# B&R Automation Studio project NewPendant_NG4_11_05_25A (part 8)

```c
					break;

			}

			if (Process[m->pCfg->HeadCfg.OSC.PROC_Indx].Param[1] == 0)
			{

				if(1)
				{

					curCalib->Points[CALIB_OSC_SFT_LIMIT].val[1] = TML_MTR_INST[m->pCfg->HeadCfg.OSC.TML_A_Indx].PosFBK + OSC_TML_Param_Set[0].MaxOscAmpl/2.0 ;

					if (m->pCfg->HeadCfg.OSC.TML_A_Indx == m->pCfg->HeadCfg.OSC.TML_B_Indx) // Only One OSC
						curCalib->Points[CALIB_OSC_SFT_LIMIT].val[3] = curCalib->Points[CALIB_OSC_SFT_LIMIT].val[1];

					strcpy(hmi->pMessage[0], " OSC Positive  ");
					strcpy(hmi->pMessage[1], " Software  ");
					strcpy(hmi->pMessage[2], " Limit SET ");
					strcpy(hmi->pMessage[3], " ");
					TimerStart(&hmi->MsgTmr, 1.5);

				}
				else
				{
					strcpy(hmi->pMessage[0], " Positive is ");
					strcpy(hmi->pMessage[1], "	 lower ");
					strcpy(hmi->pMessage[2], " than negative");
					strcpy(hmi->pMessage[3], "	TRY AGAIN ");
					TimerStart(&hmi->MsgTmr, 2.0);

				}

			}
			else
			{

				//if (TML_MTR_INST[m->pCfg->HeadCfg.OSC.TML_B_Indx].PosFBK > curCalib->Points[CALIB_OSC_SFT_LIMIT].val[2])
				if(1)
				{
					curCalib->Points[CALIB_OSC_SFT_LIMIT].val[3] = TML_MTR_INST[m->pCfg->HeadCfg.OSC.TML_B_Indx].PosFBK + OSC_TML_Param_Set[0].MaxOscAmpl/2.0;

					if (m->pCfg->HeadCfg.OSC.TML_A_Indx == m->pCfg->HeadCfg.OSC.TML_B_Indx) // Only One OSC
						curCalib->Points[CALIB_OSC_SFT_LIMIT].val[1] = curCalib->Points[CALIB_OSC_SFT_LIMIT].val[3];

					strcpy(hmi->pMessage[0], " OSC Positive  ");
					strcpy(hmi->pMessage[1], " Software  ");
					strcpy(hmi->pMessage[2], " Limit SET ");
					strcpy(hmi->pMessage[3], " ");
					TimerStart(&hmi->MsgTmr, 1.5);

				}
				else
				{
					strcpy(hmi->pMessage[0], " Positive is ");
					strcpy(hmi->pMessage[1], "	 lower ");
					strcpy(hmi->pMessage[2], " than negative");
					strcpy(hmi->pMessage[3], "	TRY AGAIN ");
					TimerStart(&hmi->MsgTmr, 2.0);

				}

			}

		break;

		/////////////////////////////////////////////////////////////////////////
		case EVNT_OSC_NEG_LIMIT_SET:

			if (m->pCfg->HeadCfg.OSC.Limits_Harcoded)
			{

				strcpy(hmi->pMessage[0], " OSC Limits  ");
				strcpy(hmi->pMessage[1], " are hardcoded  ");
				strcpy(hmi->pMessage[2], " Operation ");
				strcpy(hmi->pMessage[3], " denied");
				TimerStart(&hmi->MsgTmr, 1.5);

				break;

			}

			if((curCalib->GenSetup[SETUP_HEAD_SETUP] == BPV_v2_MT_BO_TOS)
				|| (curCalib->GenSetup[SETUP_HEAD_SETUP] == BPV_v2_TT_BO_TOS)
				|| (curCalib->GenSetup[SETUP_HEAD_SETUP] == BPV_v2_MPGH)
				|| (curCalib->GenSetup[SETUP_HEAD_SETUP] == BPV_v2_MPGV)
				 ){

					curCalib->Points[CALIB_OSC_SFT_LIMIT].val[0] = TML_MTR_INST[m->pCfg->HeadCfg.TVL.TML_Indx].PosFBK;

					strcpy(hmi->pMessage[0], " TVL (OSC) Negative  ");
					strcpy(hmi->pMessage[1], " Software  ");
					strcpy(hmi->pMessage[2], " Limit SET ");
					strcpy(hmi->pMessage[3], " ");
					TimerStart(&hmi->MsgTmr, 1.5);

					break;

			}

			if (Process[m->pCfg->HeadCfg.OSC.PROC_Indx].Param[1] == 0)
			{

				//if (TML_MTR_INST[m->pCfg->HeadCfg.OSC.TML_A_Indx].PosFBK < curCalib->Points[CALIB_OSC_SFT_LIMIT].val[1])
				if(1)
				{
					curCalib->Points[CALIB_OSC_SFT_LIMIT].val[0] = TML_MTR_INST[m->pCfg->HeadCfg.OSC.TML_A_Indx].PosFBK - OSC_TML_Param_Set[0].MaxOscAmpl/2.0;

					if (m->pCfg->HeadCfg.OSC.TML_A_Indx == m->pCfg->HeadCfg.OSC.TML_B_Indx) // Only One OSC
						curCalib->Points[CALIB_OSC_SFT_LIMIT].val[2] = curCalib->Points[CALIB_OSC_SFT_LIMIT].val[0];

					strcpy(hmi->pMessage[0], " OSC Negative  ");
					strcpy(hmi->pMessage[1], " Software  ");
					strcpy(hmi->pMessage[2], " Limit SET ");
					strcpy(hmi->pMessage[3], " ");
					TimerStart(&hmi->MsgTmr, 1.5);

				}
				else
				{
					strcpy(hmi->pMessage[0], " Negative is ");
					strcpy(hmi->pMessage[1], "	 greater ");
					strcpy(hmi->pMessage[2], " than positive");
					strcpy(hmi->pMessage[3], "	TRY AGAIN ");
					TimerStart(&hmi->MsgTmr, 2.0);

				}
			}
			else
			{

				//if (TML_MTR_INST[m->pCfg->HeadCfg.OSC.TML_B_Indx].PosFBK < curCalib->Points[CALIB_OSC_SFT_LIMIT].val[3])
				if(1)
				{
					curCalib->Points[CALIB_OSC_SFT_LIMIT].val[2] = TML_MTR_INST[m->pCfg->HeadCfg.OSC.TML_B_Indx].PosFBK - OSC_TML_Param_Set[0].MaxOscAmpl/2.0;

					if (m->pCfg->HeadCfg.OSC.TML_A_Indx == m->pCfg->HeadCfg.OSC.TML_B_Indx) // Only One OSC
						curCalib->Points[CALIB_OSC_SFT_LIMIT].val[0] = curCalib->Points[CALIB_OSC_SFT_LIMIT].val[2];

					strcpy(hmi->pMessage[0], " OSC Negative  ");
					strcpy(hmi->pMessage[1], " Software  ");
					strcpy(hmi->pMessage[2], " Limit SET ");
					strcpy(hmi->pMessage[3], " ");
					TimerStart(&hmi->MsgTmr, 1.5);

				}
				else
				{
					strcpy(hmi->pMessage[0], " Negative is ");
					strcpy(hmi->pMessage[1], "	 greater ");
					strcpy(hmi->pMessage[2], " than positive");
					strcpy(hmi->pMessage[3], "	TRY AGAIN ");
					TimerStart(&hmi->MsgTmr, 2.0);
				}

			}

		break;

		///////////////////////////////////////////////////

		case EVNT_VER_TIG_PS_CALIB:

			hmi->CalibStep = 4;
			hmi->CalibStepDone = 1;
			strcpy(hmi->pHMI_Lines[0], "Ready To Test");

			//memcpy(&hmi->tempCalib , &curCalib->Points[CALIB_TIG_AMPS_CMD] , sizeof(tempCalib));
		break;

		case EVNT_VER_HW_PS_CALIB:

			hmi->CalibStep = 4;
			hmi->CalibStepDone = 1;
			strcpy(hmi->pHMI_Lines[0], "Ready To Test");

			//memcpy(&hmi->tempCalib , &curCalib->Points[CALIB_HW_AMPS_CMD] , sizeof(tempCalib));
		break;

		case EVNT_VER_TVL_CALIB:

			hmi->CalibStep = 6;
			hmi->CalibStepDone = 1;
			strcpy(hmi->pHMI_Lines[0], "Ready To Test");

			//memcpy(&hmi->tempCalib , &curCalib->Points[CALIB_TVL_SPEED_CMD] , sizeof(tempCalib));
		break;

		case EVNT_VER_WF_CALIB:

			hmi->CalibStep = 6;
			hmi->CalibStepDone = 1;
			strcpy(hmi->pHMI_Lines[0], "Ready To Test");

			//memcpy(&hmi->tempCalib , &curCalib->Points[CALIB_WF_SPEED_CMD] , sizeof(tempCalib));
		break;

		////////////////////////////////////////////////////////////////////
		case EVNT_SAVE_SETUP_BIN:

			if (File_RW.CMD == 0)
			{
				File_RW.CMD 		= F_SAVE_SETUP_BIN;

				strcpy(hmi->pMessage[0], " Setup As Binary");
				strcpy(hmi->pMessage[1], "");
				strcpy(hmi->pMessage[2], "	   SAVED ");
				strcpy(hmi->pMessage[3], " ");
				TimerStart(&hmi->MsgTmr, 1.0);

			}

		break;

		case EVNT_SAVE_SETUP_AS_BIN:

			if (File_RW.CMD == 0)
			{

				if (strlen(curCfg->CurProgramName) == 0)
					strcpy(curCfg->CurProgramName, "Default");

				strcpy(File_RW.fileNewName, curCfg->CurProgramName);

				if(Find_ext_txt(File_RW.fileNewName , "_state"))
					File_RW.fileNewName[strlen(File_RW.fileNewName) - 6] = 0;

				if(Find_ext_txt(File_RW.fileNewName , "_calib"))
					File_RW.fileNewName[strlen(File_RW.fileNewName) - 6] = 0;

				if(!Find_ext_txt(File_RW.fileNewName , "_setup"))
					strcat(File_RW.fileNewName, "_setup");

				File_RW.CMD = F_SAVE_AS_CURCFG_BIN;

				strcpy(hmi->pMessage[0], " Setup ");
				strcpy(hmi->pMessage[1], " As Binary ");
				strcpy(hmi->pMessage[2], "	   SAVED ");
				strcpy(hmi->pMessage[3], " ");
				TimerStart(&hmi->MsgTmr, 1.0);

			}

		break;

		case EVNT_SAVE_FULL_AS_BIN:

			if (File_RW.CMD == 0)
			{

				if (strlen(curCfg->CurProgramName) == 0)
					strcpy(curCfg->CurProgramName, "Default");

				strcpy(File_RW.fileNewName, curCfg->CurProgramName);

				if(Find_ext_txt(File_RW.fileNewName , "_setup"))
					File_RW.fileNewName[strlen(File_RW.fileNewName) - 6] = 0;

				if(Find_ext_txt(File_RW.fileNewName , "_calib"))
					File_RW.fileNewName[strlen(File_RW.fileNewName) - 6] = 0;

				if(!Find_ext_txt(File_RW.fileNewName , "_state"))
					strcat(File_RW.fileNewName, "_state");

				File_RW.CMD = F_SAVE_AS_FULL_BIN;

				strcpy(hmi->pMessage[0], "Machine State");
				strcpy(hmi->pMessage[1], " As Binary ");
				strcpy(hmi->pMessage[2], "	   SAVED ");
				strcpy(hmi->pMessage[3], " ");
				TimerStart(&hmi->MsgTmr, 1.0);

			}

		break;

		case EVNT_SAVE_CALIB_AS_BIN:

			if (File_RW.CMD == 0)
			{

				if (strlen(curCfg->CurProgramName) == 0)
					strcpy(curCfg->CurProgramName, "Default");

				strcpy(File_RW.fileNewName, curCfg->CurProgramName);

				if(Find_ext_txt(File_RW.fileNewName , "_setup"))
					File_RW.fileNewName[strlen(File_RW.fileNewName) - 6] = 0;

				if(Find_ext_txt(File_RW.fileNewName , "_state"))
					File_RW.fileNewName[strlen(File_RW.fileNewName) - 6] = 0;

				if(!Find_ext_txt(File_RW.fileNewName , "_calib"))
					strcat(File_RW.fileNewName, "_calib");

				File_RW.CMD = F_SAVE_AS_CALIB_BIN;

				strcpy(hmi->pMessage[0], " Calibration");
				strcpy(hmi->pMessage[1], " As Binary ");
				strcpy(hmi->pMessage[2], "	   SAVED ");
				strcpy(hmi->pMessage[3], " ");
				TimerStart(&hmi->MsgTmr, 1.0);

			}

		break;

	}

	// Temporary Patch it should be on event process switch
	if ((intrf->WheelDelta != 0) || ((intrf->GlblBtnCmd[0] &ANDR_BTN_RIGHT) && !intrf->_intr._GlblBtnCmd[0]) ||
	((intrf->GlblBtnCmd[0] &ANDR_BTN_LEFT) && !intrf->_intr._GlblBtnCmd[0]))
	{
		if (curCfg->Param_ENUM[parENUM_WF_WP_Relation].val[0] > 0)
		{
			for (i = 0; i < m->numZone; i++)
			curCfg->Param[parWP_SpeedSP].val[i] = curCfg->Param[parWF_SpeedSP].val[i] *0.31552314834734205493308631414126;
		}

	}

// Check Updated Values
	if(hmi->PleaseUpdate)
	{

		if (!intrf->TickPlus && !intrf->TickMinus && !hmi->BypassTicks)
			return;

		curCfg->Dirty		= 1;

		if (!m->pScaledVar)
		return;

		pVar =(Scaled_Var_obj *)m->pScaledVar;

		//seg = pVar[indx].segm;
		//seg = 0;
		seg = (hmi->PleaseUpdate & 0xFC00) / 1024;

		if ((! (curCalib->GenSetup[SETUP_WHERE_FILL] == 1) && (hmi->curHeadID == 65535))) //Not only Keyboard && Segment Page
		Fill_Segments(curCfg, hmi->PleaseUpdate & 0x3FF, seg, curCalib->GenSetup[SETUP_AUTO_FILL], m->sm.Step);

		switch (hmi->PleaseUpdate & 0x3FF)
		{
			///// Test /////////

			/*
			case parTIG_AmpSP:

				strcpy(hmi->pMessage[0], " TIG Amplit  ");
				xsprintf(hmi->pMessage[1] , "Segm: %d" , seg);
				strcpy(hmi->pMessage[2], " nic");
				strcpy(hmi->pMessage[3], " test");
				TimerStart(&hmi->MsgTmr, 1.5);

			break;
			*/

			///////////////////////////
			case parWF_SpeedSP:

				if (curCfg->Param_ENUM[parENUM_WF_WP_Relation].val[0] > 0)
				{
					for (i = 0; i < m->numZone; i++)
						curCfg->Param[parWP_SpeedSP].val[i] = curCfg->Param[parWF_SpeedSP].val[i] *0.31552314834734205493308631414126;
				}

			break;

			case parOSC_InitAmplit:

				/*

				if(curCfg->Param[parOSC_InitAmplit].val[seg] > curCfg->Param[parOSC_Amplit].val[seg] ){

					curCfg->Param[parOSC_InitAmplit].val[seg] = curCfg->Param[parOSC_Amplit].val[seg];

					strcpy(hmi->pMessage[0], " OSC Init   ");
					strcpy(hmi->pMessage[1], " Amplitude ");
					strcpy(hmi->pMessage[2], " bigger then ");
					strcpy(hmi->pMessage[3], " Primery Amplitude");
					TimerStart(&hmi->MsgTmr, 1.5);

				}
				*/
			break;

			case parOSC_FinalAmplit:

				/*

				if(curCfg->Param[parOSC_FinalAmplit].val[seg] > curCfg->Param[parOSC_Amplit].val[seg] ){

					curCfg->Param[parOSC_FinalAmplit].val[seg] = curCfg->Param[parOSC_Amplit].val[seg];

					strcpy(hmi->pMessage[0], " OSC Final   ");
					strcpy(hmi->pMessage[1], " Amplitude ");
					strcpy(hmi->pMessage[2], " bigger then ");
					strcpy(hmi->pMessage[3], " Primery Amplitude");
					TimerStart(&hmi->MsgTmr, 1.5);

				}
				*/
			break;

			case parOSC_Amplit:
				Check_parOSC_Amplit(curCfg, hmi, seg);

				/*
				if(curCfg->Param[parOSC_Amplit].val[seg] < curCfg->Param[parOSC_FinalAmplit].val[seg] ){

					curCfg->Param[parOSC_Amplit].val[seg] = curCfg->Param[parOSC_FinalAmplit].val[seg];

					strcpy(hmi->pMessage[0], " OSC Primery	 ");
					strcpy(hmi->pMessage[1], " Amplitude ");
					strcpy(hmi->pMessage[2], " smaller then ");
					strcpy(hmi->pMessage[3], " Final Amplitude");
					TimerStart(&hmi->MsgTmr, 1.5);

				}

				if(curCfg->Param[parOSC_Amplit].val[seg] < curCfg->Param[parOSC_InitAmplit].val[seg] ){

					curCfg->Param[parOSC_Amplit].val[seg] = curCfg->Param[parOSC_InitAmplit].val[seg];

					strcpy(hmi->pMessage[0], " OSC Primery	 ");
					strcpy(hmi->pMessage[1], " Amplitude ");
					strcpy(hmi->pMessage[2], " smaller then ");
					strcpy(hmi->pMessage[3], " Init Amplitude");
					TimerStart(&hmi->MsgTmr, 1.5);

				}

				if(curCfg->Param[parOSC_Excur].val[seg] > 0 ){

					x = curCfg->Param[parOSC_Amplit].val[seg] / curCfg->Param[parOSC_Excur].val[seg];

					if(x > curCfg->Param[parOSC_MaxTvlVel].val[0] ){

						curCfg->Param[parOSC_Amplit].val[seg] = curCfg->Param[parOSC_MaxTvlVel].val[0] * curCfg->Param
					[parOSC_Excur].val[seg];

						strcpy(hmi->pMessage[0], " OSC	 ");
						strcpy(hmi->pMessage[1], " Amplitude ");
						strcpy(hmi->pMessage[2], " was");
						strcpy(hmi->pMessage[3], " too high");
						TimerStart(&hmi->MsgTmr, 1.5);

					}

				}

				*/
			break;

			case parOSC_Excur:

				Check_parOSC_Excur(curCfg, hmi, seg);

				/*

				if((curCfg->Param[parOSC_Excur].val[seg] > 0)
					&& (curCfg->Param[parOSC_MaxTvlVel].val[0] > 0)){

					x = curCfg->Param[parOSC_Amplit].val[seg] / curCfg->Param[parOSC_Excur].val[seg];

					if(x >curCfg->Param[parOSC_MaxTvlVel].val[0] ){

						curCfg->Param[parOSC_Excur].val[seg] = curCfg->Param[parOSC_Amplit].val[seg] /		curCfg->Param
					[parOSC_MaxTvlVel].val[0];

						strcpy(hmi->pMessage[0], " OSC	 ");
						strcpy(hmi->pMessage[1], " Excurtion ");
						strcpy(hmi->pMessage[2], " was");
						strcpy(hmi->pMessage[3], " too small");
						TimerStart(&hmi->MsgTmr, 1.5);

					}

				}

				*/
			break;

			case parTVL_InitVel:

			if (curCfg->Param[parTVL_InitVel].val[0] > curCfg->Param[parTVL_VelSP].val[seg])
			{
				curCfg->Param[parTVL_InitVel].val[0] = curCfg->Param[parTVL_VelSP].val[seg];

				strcpy(hmi->pMessage[0], " TVL Init   ");
				strcpy(hmi->pMessage[1], " Speed ");
				strcpy(hmi->pMessage[2], " bigger then ");
				strcpy(hmi->pMessage[3], " Primery Speed");
				TimerStart(&hmi->MsgTmr, 1.5);

			}

			break;

			case parTVL_FinalVel:

				if (curCfg->Param[parTVL_FinalVel].val[0] > curCfg->Param[parTVL_VelSP].val[seg])
				{
					curCfg->Param[parTVL_FinalVel].val[0] = curCfg->Param[parTVL_VelSP].val[seg];

					strcpy(hmi->pMessage[0], " TVL Final   ");
					strcpy(hmi->pMessage[1], " Speed ");
					strcpy(hmi->pMessage[2], " bigger then ");
					strcpy(hmi->pMessage[3], " Primery Speed");
					TimerStart(&hmi->MsgTmr, 1.5);
				}

			break;

			case parTVL_VelSP:

				if (curCfg->Param[parTVL_VelSP].val[seg] < curCfg->Param[parTVL_InitVel].val[0])
				{
					curCfg->Param[parTVL_VelSP].val[seg] = curCfg->Param[parTVL_InitVel].val[0];

					strcpy(hmi->pMessage[0], " TVL Primery	 ");
					strcpy(hmi->pMessage[1], " Speed ");
					strcpy(hmi->pMessage[2], " smaller then ");
					strcpy(hmi->pMessage[3], " Init Speed");
					TimerStart(&hmi->MsgTmr, 1.5);

				}

				if (curCfg->Param[parTVL_VelSP].val[seg] < curCfg->Param[parTVL_FinalVel].val[0])
				{
					curCfg->Param[parTVL_VelSP].val[seg] = curCfg->Param[parTVL_FinalVel].val[0];

					strcpy(hmi->pMessage[0], " TVL Primery	 ");
					strcpy(hmi->pMessage[1], " Speed ");
					strcpy(hmi->pMessage[2], " smaller then ");
					strcpy(hmi->pMessage[3], " Final Speed");
					TimerStart(&hmi->MsgTmr, 1.5);

				}

			break;

			case parAVC_FbkFilter:

				TML_MTR_INST[m->pCfg->HeadCfg.AVC.TML_A_Indx]._cfg.signFilter =	curCfg->Param[parAVC_FbkFilter].val[0];
				VectorStateMach[VECT_AVC].xCMD = VECT_UpdateSignFilter;

			break;

			case parAVC_DB_Window:

				VectorStateMach[VECT_AVC].fParam[0] = curCfg->Param[parAVC_DB_Window].val[0];
				VectorStateMach[VECT_AVC].xCMD = VECT_Set_MaxError;

			break;

			case parAVC_KIP:
			case parAVC_KPP:

				TML_MTR_INST[m->pCfg->HeadCfg.AVC.TML_A_Indx]._cfg.kpp = (DINT)(curCfg->Param[parAVC_KPP].val[0] *TML_MTR_INST[m->pCfg->HeadCfg.AVC.TML_A_Indx]._cfg.kppMax);
				TML_MTR_INST[m->pCfg->HeadCfg.AVC.TML_A_Indx]._cfg.kip = (DINT)(curCfg->Param[parAVC_KIP].val[0] *TML_MTR_INST[m->pCfg->HeadCfg.AVC.TML_A_Indx]._cfg.kipMax);

				VectorStateMach[VECT_AVC].xCMD = VECT_Set_PID_Param;

				TML_MTR_INST[m->pCfg->HeadCfg.AVC.TML_B_Indx]._cfg.kpp = (DINT)(curCfg->Param[parAVC_KPP].val[0] *TML_MTR_INST[m->pCfg->HeadCfg.AVC.TML_A_Indx]._cfg.kppMax);
				TML_MTR_INST[m->pCfg->HeadCfg.AVC.TML_B_Indx]._cfg.kip = (DINT)(curCfg->Param[parAVC_KIP].val[0] *TML_MTR_INST[m->pCfg->HeadCfg.AVC.TML_A_Indx]._cfg.kipMax);

				VectorStateMach[VECT_AVC2].xCMD = VECT_Set_PID_Param;

			break;

			case parTVL_RunDist:

				PleaseUpdateHeadSetup(m);

			break;

			case parTVL_TrackDia:

			break;

		}

		////////   Parameter Leaders /////////////////////

		if (hmi->curNodeID == P_PARAM_WELD)
		{

			switch (indx)
			{
				case parAVC_Upslope:
				break;

				case parWF_RampUp:
				break;

				case parWF_RampDwn:
				break;

				case parAVC_DownSlope:
				break;
			}

		}
	}

	hmi->FiredEvent = 0;

}

void EditParam(UINT paramIndx)
{

	if (hmi->curNodeID >= P_MENU)
	{
		strcpy(hmi->ActiveBanner, "");
		return;
	}

	GlblBtnLED_Mask 	= intrf->GlblBtnCmd[0];

	Force_ENTR_LCD		= 1;
	hmi->DynPageNodeIndx = P_POP_UP;

	nodes[P_POP_UP].var.Var1ID = paramIndx;

	if (curCfg->Param[paramIndx].segmYes)
		var[paramIndx].segm = m->curSegm[ZONE];

	return;

}

void JogProcessAndroid(HMI_INTRF_typ * intrf, UINT procIndx, float gain)
{

	Process[procIndx].xCMD = prcsDirectCntrl;
	Process[procIndx].fParam[0] = gain;

	return;
}

void TakeNextWeldProgram(HMI_typ * hmi)
{

	if((strlen(curCfg->NextProgramName) > 31)
		|| (strlen(curCfg->NextProgramName) == 0))
		strcpy(curCfg->NextProgramName, PRG_NO_NEXT);

	//if (strlen(curCfg->NextProgramName) && strcmp(curCfg->NextProgramName, PRG_NO_NEXT))
	if(strcmp(curCfg->NextProgramName, PRG_NO_NEXT))
	{

		strcpy(File_RW.deviceName, "WeldPrograms");

		strcpy(File_RW.fileName, curCfg->NextProgramName);

		DeleteExtension(File_RW.fileName);

		if (File_RW.Mode == F_MODE_XML)
			strcat(File_RW.fileName, PRG_FILE_EXT);

		File_RW.CMD 		= F_LOAD_CURCFG;

		if (curCfg->Dirty)
		{
			strcpy(hmi->pMessage[0], "Changes are LOST !!!");
			xsprintf(hmi->pMessage[1], " %s", File_RW.fileName);
			strcpy(hmi->pMessage[2], "	is");
			strcpy(hmi->pMessage[3], " Loaded ");
			TimerStart(&hmi->MsgTmr, 1.0);
		}
		else
		{
			strcpy(hmi->pMessage[0], " NEXT Program ");
			xsprintf(hmi->pMessage[1], " %s", File_RW.fileName);
			strcpy(hmi->pMessage[2], "	is");
			strcpy(hmi->pMessage[3], " Loaded ");
			TimerStart(&hmi->MsgTmr, 1.0);
		}

	}

}

void AndroidHelper(MASTER_typ * m, UINT n)
{

	if (!m || n > 1)
		return;

	/*
	m->AndIntrf[n].MasterMode = m->Mode;

	switch(m->AndIntrf[n].UserLevel){

	case USER_OPERATOR: strcpy(m->AndIntrf[n].UserLevelTXT , "OPERATOR"); break;

	case USER_ADJUSTER: strcpy(m->AndIntrf[n].UserLevelTXT , "ADJUSTER"); break;

	case USER_MANAGER:	strcpy(m->AndIntrf[n].UserLevelTXT , "MANAGER"); break;

	case USER_JA:		strcpy(m->AndIntrf[n].UserLevelTXT , "DESIGNER"); break;

	default: strcpy(m->AndIntrf[n].UserLevelTXT , "WRONG LEVEL"); break;

	}

	switch(m->AndIntrf[n].MasterMode){

	case MASTER_MODE_STOP: strcpy(m->AndIntrf[n].MasterModTXT , "IDLE"); break;

	case MASTER_MODE_RUN: strcpy(m->AndIntrf[n].MasterModTXT , "RUN"); break;

	case MASTER_MODE_CALIB_STOP:	strcpy(m->AndIntrf[n].MasterModTXT , "CALIBR. IDLE"); break;

	case MASTER_MODE_CALIB_RUN:	strcpy(m->AndIntrf[n].MasterModTXT , "CALIBR. RUN"); break;

	case MASTER_MODE_ERROR:			strcpy(m->AndIntrf[n].MasterModTXT , "ERROR"); break;

	case MASTER_MODE_ESTOP: 		strcpy(m->AndIntrf[n].MasterModTXT , "ESTOP"); break;

	default: strcpy(m->AndIntrf[n].MasterModTXT , "INITIAL"); break;

	}

	*/
}

void StopModeAndroidButtons(MASTER_typ * m, HMI_typ * hmi, HMI_INTRF_typ * intrf, LCD_MGR_obj * lcd)
{
	UINT			i;
	UINT			par;
	CurCfg_typ *	curCfg;

	curCfg				= m->pCurCfg;

	if (!curCfg)
		return;

	////////////
	switch (intrf->GlblBtnCmd[0])
	{
		case ANDR_BTN_HOME:

		break;

		case ANDR_BTN_ARC_AMPS_NEG:

			if (m->AndIntrf[0].GlblBtnLED[1] &0x2){

					strcpy(hmi->ActiveBanner, "WB#1 JOG REV");
					JogProcessAndroid(intrf, m->pCfg->HeadCfg.WB[WB_UD].PROC_Indx,(-1.0));

			}else if(!Process[PROC_INDX].Disable){

				switch(curCalib->GenSetup[SETUP_HEAD_SETUP]){

					case BPV_v2:
					case BPV_v2_Video:
					case BPV_v2_MPBO:
					case BPV_v2_MPGV:
					case BPV_v2_MPGH:
					//dodane 6Dec23
					case BPV_v2_MT:

						strcpy(hmi->ActiveBanner, " INDX JOG DWN ");

						JogProcessAndroid(intrf, m->pCfg->HeadCfg.INDX.PROC_Indx,
						m->pCfg->HeadCfg.INDX.BtnJog_Gain * getBtnProgress () * (-1.0));

					break;

					case BPV_v2_MT_BO:
					case BPV_v2_MT_BO_TOS:
					case BPV_v2_TT_BO:
					case BPV_v2_TT_BO_TOS:

						strcpy(hmi->ActiveBanner, "INDEX Not installed ");

					break;

					default:

						strcpy(hmi->ActiveBanner, "INDEX JOG REV ");

						if(hmi->curHeadID != P_MODE_INDX_CALIB)
							Process[m->pCfg->HeadCfg.INDX.PROC_Indx].Param[3] = 0; // Both head Jogging

						Process[m->pCfg->HeadCfg.INDX.PROC_Indx].xCMD = prcsJOGpos;
						Process[m->pCfg->HeadCfg.INDX.PROC_Indx].fParam[0] = (-1.0);

					break;

				}

			}
			else{

				strcpy(hmi->ActiveBanner, "INDEX Process Disabled ");

			}

		break;

		case ANDR_BTN_ARC_AMPS_POS:

			if (m->AndIntrf[0].GlblBtnLED[1] &0x2){

				strcpy(hmi->ActiveBanner, "WB#1 JOG FWD");
				JogProcessAndroid(intrf, m->pCfg->HeadCfg.WB[WB_UD].PROC_Indx,(1.0));

			}else if(!Process[PROC_INDX].Disable){

				switch(curCalib->GenSetup[SETUP_HEAD_SETUP]){

					case BPV_v2:
					case BPV_v2_Video:
					case BPV_v2_MPBO:
					case BPV_v2_MPGV:
					case BPV_v2_MPGH:
					//dodane 6Dec23
					case BPV_v2_MT:

						strcpy(hmi->ActiveBanner, " INDX JOG UP ");

						JogProcessAndroid(intrf, m->pCfg->HeadCfg.INDX.PROC_Indx,
						m->pCfg->HeadCfg.INDX.BtnJog_Gain * getBtnProgress ());

					break;

					case BPV_v2_MT_BO:
					case BPV_v2_MT_BO_TOS:
					case BPV_v2_TT_BO:
					case BPV_v2_TT_BO_TOS:

						strcpy(hmi->ActiveBanner, "INDEX Not installed ");

					break;

					default:

						strcpy(hmi->ActiveBanner, "INDEX JOG FWD ");

						if(hmi->curHeadID != P_MODE_INDX_CALIB)
							Process[m->pCfg->HeadCfg.INDX.PROC_Indx].Param[3] = 0; // Both head Jogging

						Process[m->pCfg->HeadCfg.INDX.PROC_Indx].xCMD = prcsJOGpos;
						Process[m->pCfg->HeadCfg.INDX.PROC_Indx].fParam[0] = 1.0;

					break;

				}

			}
			else{

				strcpy(hmi->ActiveBanner, "INDEX Process Disabled ");

			}

		break;

		case ANDR_BTN_TRAVEL_SPEED_NEG:

			if (m->AndIntrf[0].GlblBtnLED[1] &0x2){

				strcpy(hmi->ActiveBanner, "WB#2 JOG REV");
				JogProcessAndroid(intrf, m->pCfg->HeadCfg.WB[WB_LR].PROC_Indx,(-1.0));

			}else{

				strcpy(hmi->ActiveBanner, " TRAVEL JOG REV ");
				JogProcessAndroid(intrf, m->pCfg->HeadCfg.TVL.PROC_Indx,
				m->pCfg->HeadCfg.TVL.BtnJog_Gain * getBtnProgress() * (-1.0));

				if (_TVL_Latch_Latched && TVL_Latch_Latched)
				{
					TVL_Latch_Latched	= 0;
					_TVL_Latch_Latched	= TVL_Latch_Latched;
					TVL_Latch_Cnt		= 0;
				}

				if (!TVL_Latch_Latched)
				{
					if (TVL_Latch_Cnt < TVL_Latch_Tm)
						TVL_Latch_Cnt++;
					else
						TVL_Latch_Latched = 1;
				}

			}

		break;

		case ANDR_BTN_TRAVEL_SPEED_POS:

			if (m->AndIntrf[0].GlblBtnLED[1] &0x2){

				strcpy(hmi->ActiveBanner, "WB#2 JOG FWD");
				JogProcessAndroid(intrf, m->pCfg->HeadCfg.WB[WB_LR].PROC_Indx,(1.0));

			}else{

				strcpy(hmi->ActiveBanner, " TRAVEL JOG FWD");
				JogProcessAndroid(intrf, m->pCfg->HeadCfg.TVL.PROC_Indx,
				m->pCfg->HeadCfg.TVL.BtnJog_Gain * getBtnProgress());

				if (_TVL_Latch_Latched && TVL_Latch_Latched)
				{
					TVL_Latch_Latched	= 0;
					_TVL_Latch_Latched	= TVL_Latch_Latched;
					TVL_Latch_Cnt		= 0;
				}

				if (!TVL_Latch_Latched)
				{
					if (TVL_Latch_Cnt < TVL_Latch_Tm)
						TVL_Latch_Cnt++;
					else
						TVL_Latch_Latched = 2;
				}

			}

		break;

		case ANDR_BTN_WIRE_SPEED_NEG:

			if (m->AndIntrf[0].GlblBtnLED[1] &0x2){

				///  LAMPS ON / OFF
				if (!intrf->_intr._GlblBtnCmd[0]){
					Hardware[1].Outp[9] = !Hardware[1].Outp[9];

					if(Hardware[1].Outp[9]){

						/* was only for Super Mini Head

						if(VectorStateMach[m->pCfg->HeadCfg.OSC.VECT_A_Indx].xCMD == 0)
							VectorStateMach[m->pCfg->HeadCfg.OSC.VECT_A_Indx].xCMD = VECT_Set_OUT0;

						if(VectorStateMach[m->pCfg->HeadCfg.WF.VECT_A_Indx].xCMD == 0)
							VectorStateMach[m->pCfg->HeadCfg.WF.VECT_A_Indx].xCMD = VECT_Set_OUT0;

						*/

						if(m->pCfg->HeadCfg.LampOnOFF.VECT_A_Indx > 0){ // Zero means - do not apply

							if(VectorStateMach[m->pCfg->HeadCfg.LampOnOFF.VECT_A_Indx - 1].xCMD == 0)
								VectorStateMach[m->pCfg->HeadCfg.LampOnOFF.VECT_A_Indx -1].xCMD = VECT_Set_OUT0;

						}

						if(m->pCfg->HeadCfg.LampOnOFF.VECT_B_Indx > 0){ // Zero means - do not apply

							if(VectorStateMach[m->pCfg->HeadCfg.LampOnOFF.VECT_B_Indx-1].xCMD == 0)
								VectorStateMach[m->pCfg->HeadCfg.LampOnOFF.VECT_B_Indx-1].xCMD = VECT_Set_OUT0;

						}

					}
					else{

						if(m->pCfg->HeadCfg.LampOnOFF.VECT_A_Indx > 0){ // Zero means - do not apply

							if(VectorStateMach[m->pCfg->HeadCfg.LampOnOFF.VECT_A_Indx - 1].xCMD == 0)
								VectorStateMach[m->pCfg->HeadCfg.LampOnOFF.VECT_A_Indx -1].xCMD = VECT_Rst_OUT0;

						}

						if(m->pCfg->HeadCfg.LampOnOFF.VECT_B_Indx > 0){ // Zero means - do not apply

							if(VectorStateMach[m->pCfg->HeadCfg.LampOnOFF.VECT_B_Indx-1].xCMD == 0)
								VectorStateMach[m->pCfg->HeadCfg.LampOnOFF.VECT_B_Indx-1].xCMD = VECT_Rst_OUT0;

						}

						/* was only for Super Mini Head
						if(VectorStateMach[m->pCfg->HeadCfg.OSC.VECT_A_Indx].xCMD == 0)
							VectorStateMach[m->pCfg->HeadCfg.OSC.VECT_A_Indx].xCMD = VECT_Rst_OUT0;

						if(VectorStateMach[m->pCfg->HeadCfg.WF.VECT_A_Indx].xCMD == 0)
							VectorStateMach[m->pCfg->HeadCfg.WF.VECT_A_Indx].xCMD = VECT_Rst_OUT0;
						*/

					}

				}

			}else{

				strcpy(hmi->ActiveBanner, "WIRE JOG REV");
				JogProcessAndroid(intrf, m->pCfg->HeadCfg.WF.PROC_Indx,
				m->pCfg->HeadCfg.WF.BtnJog_Gain * getBtnProgress() * (-1.0));

			}

		break;

		case ANDR_BTN_WIRE_SPEED_POS:

			if (m->AndIntrf[0].GlblBtnLED[1] &0x2){

				// Camera View
				if (!intrf->_intr._GlblBtnCmd[0])
					MV[0].xCMD = MV_LOAD_NEXT_CMD;

			}else{

				strcpy(hmi->ActiveBanner, "WIRE JOG FWD");
				JogProcessAndroid(intrf, m->pCfg->HeadCfg.WF.PROC_Indx,
				m->pCfg->HeadCfg.WF.BtnJog_Gain * getBtnProgress());

			}

		break;

		case ANDR_BTN_AVC_VOLTS_NEG:

			strcpy(hmi->ActiveBanner, " AVC JOG DOWN ");
			JogProcessAndroid(intrf, m->pCfg->HeadCfg.AVC.PROC_Indx,
			m->pCfg->HeadCfg.AVC.BtnJog_Gain * getBtnProgress() * (-1.0));

		break;

		case ANDR_BTN_AVC_VOLTS_POS:

			strcpy(hmi->ActiveBanner, " AVC JOG UP ");
			JogProcessAndroid(intrf, m->pCfg->HeadCfg.AVC.PROC_Indx,
			m->pCfg->HeadCfg.AVC.BtnJog_Gain * getBtnProgress());

		break;

		case ANDR_BTN_OSC_SPEED_NEG:

			if (Process[m->pCfg->HeadCfg.OSC.PROC_Indx].Status == prcsSTATUS_Run)
			{
				strcpy(hmi->ActiveBanner, "OSC	TIME Minus");

				if (m->AndIntrf[0].GlblBtnLED[1] &0x1)
					par = parOSC_Dwell_In;

				else if (m->AndIntrf[0].GlblBtnLED[1] &0x2)
					par = parOSC_Dwell_Out;

				else
					par = parOSC_Excur;

				if (!intrf->_intr._GlblBtnCmd[0])
				{
					DecrParam(curCfg, par, m->curSegm[ZONE], 1.0);

					if (par == parOSC_Excur)
						Check_parOSC_Excur(curCfg, hmi, m->curSegm[ZONE]);

					if (! (curCalib->GenSetup[SETUP_WHERE_FILL] == 2)) //Not only Editor
						Fill_Segments(curCfg, par, m->curSegm[ZONE], curCalib->GenSetup[SETUP_AUTO_FILL], m->sm.Step);

				}

			}
			else if(!Process[PROC_WRST].Disable){

				switch(curCalib->GenSetup[SETUP_HEAD_SETUP]){

					/*
					case BPV_v2:
					case BPV_v2_MPBO:
					case BPV_v2_MPGV:
					case BPV_v2_MPGH:

						strcpy(hmi->ActiveBanner, " INDX JOG DWN ");

						JogProcessAndroid(intrf, m->pCfg->HeadCfg.INDX.PROC_Indx,
						m->pCfg->HeadCfg.INDX.BtnJog_Gain * getBtnProgress () * (-1.0));

					break;
					*/

					case BPV_v2:
					case BPV_v2_Video:
					case BPV_v2_MPBO:
					case BPV_v2_MPGV:
					case BPV_v2_MPGH:
					case BPV_v2_MT_BO:
					case BPV_v2_MT_BO_TOS:
					case BPV_v2_TT_BO:
					case BPV_v2_TT_BO_TOS:
					//dodane 6Dec23
					case BPV_v2_MT:

						strcpy(hmi->ActiveBanner, " WRST JOG Left ");

						Process[m->pCfg->HeadCfg.WRST.PROC_Indx].xCMD = prcsJOGpos;
						Process[m->pCfg->HeadCfg.WRST.PROC_Indx].fParam[0] = m->pCfg->HeadCfg.WRST.BtnJog_Gain * getBtnProgress () * (-1.0);

					break;

					default:

						strcpy(hmi->ActiveBanner, "WRST JOG Left");

						JogProcessAndroid(intrf, m->pCfg->HeadCfg.WRST.PROC_Indx,
						m->pCfg->HeadCfg.WRST.BtnJog_Gain * getBtnProgress () * (-1.0));

					break;

				}

			}
			else{

				strcpy(hmi->ActiveBanner, "WRST Process Disabled ");

			}

		break;

		case ANDR_BTN_OSC_SPEED_POS:

			if (Process[m->pCfg->HeadCfg.OSC.PROC_Indx].Status == prcsSTATUS_Run)
			{

				strcpy(hmi->ActiveBanner, "OSC	TIME plus");

				if (m->AndIntrf[0].GlblBtnLED[1] &0x1)
					par = parOSC_Dwell_In;

				else if (m->AndIntrf[0].GlblBtnLED[1] &0x2)
					par = parOSC_Dwell_Out;

				else
					par = parOSC_Excur;

				if (!intrf->_intr._GlblBtnCmd[0])
				{
					IncrParam(curCfg, par, m->curSegm[ZONE], 1.0);

					if (par == parOSC_Excur)
						Check_parOSC_Excur(curCfg, hmi, m->curSegm[ZONE]);

					if (! (curCalib->GenSetup[SETUP_WHERE_FILL] == 2)) //Not only Editor
						Fill_Segments(curCfg, par, m->curSegm[ZONE], curCalib->GenSetup[SETUP_AUTO_FILL], m->sm.Step);
				}
			}
			else if(!Process[PROC_WRST].Disable){

				switch(curCalib->GenSetup[SETUP_HEAD_SETUP]){

					/*
					case BPV_v2:
					case BPV_v2_MPBO:
					case BPV_v2_MPGV:
					case BPV_v2_MPGH:

						strcpy(hmi->ActiveBanner, " INDX JOG UP ");

						JogProcessAndroid(intrf, m->pCfg->HeadCfg.INDX.PROC_Indx,
						m->pCfg->HeadCfg.INDX.BtnJog_Gain * getBtnProgress ());

					break;
					*/

					case BPV_v2:
					case BPV_v2_Video:
					case BPV_v2_MPBO:
					case BPV_v2_MPGV:
					case BPV_v2_MPGH:
					case BPV_v2_MT_BO:
					case BPV_v2_MT_BO_TOS:
					case BPV_v2_TT_BO:
					case BPV_v2_TT_BO_TOS:
					//dodane 6Dec23
					case BPV_v2_MT:

						strcpy(hmi->ActiveBanner, " WRST JOG Right  ");

						Process[m->pCfg->HeadCfg.WRST.PROC_Indx].xCMD = prcsJOGpos;
						Process[m->pCfg->HeadCfg.WRST.PROC_Indx].fParam[0] = m->pCfg->HeadCfg.WRST.BtnJog_Gain * getBtnProgress ();
					break;

					default:

						strcpy(hmi->ActiveBanner, " WRST JOG Right ");

						JogProcessAndroid(intrf, m->pCfg->HeadCfg.WRST.PROC_Indx,
						m->pCfg->HeadCfg.WRST.BtnJog_Gain * getBtnProgress ());

					break;

				}

			}
			else{

				strcpy(hmi->ActiveBanner, "WRST Process Disabled ");

			}

		break;

		case ANDR_BTN_OSC_AMPL_NEG:

			if (Process[m->pCfg->HeadCfg.OSC.PROC_Indx].Status == prcsSTATUS_Run)
			{
				strcpy(hmi->ActiveBanner, "BTN_OSC_AMPL_NEG ");

				if (!intrf->_intr._GlblBtnCmd[0])
					DecrParam(curCfg, parOSC_Amplit, m->curSegm[ZONE], 1.0);

				Check_parOSC_Amplit(curCfg, hmi, m->curSegm[0]);
			}
			else if ((Process[m->pCfg->HeadCfg.OSC.PROC_Indx].Status == prcsSTATUS_Stopped) ||
			(Process[m->pCfg->HeadCfg.OSC.PROC_Indx].Status == prcsSTATUS_DirectCntrl))
			{
				strcpy(hmi->ActiveBanner, "OSC JOG LEFT");

				switch (m->pCfg->HeadCfg.OSC.BtnJog_Mode)
				{
					case BTN_JOG_MODE_SINGLE:

						JogProcessAndroid(intrf, m->pCfg->HeadCfg.OSC.PROC_Indx,
						m->pCfg->HeadCfg.OSC.BtnJog_Gain * getBtnProgress () * (-1.0));

					break;

					case BTN_JOG_MODE_DUAL:

						if (m->ToolHeadID)
							JogProcessAndroid(intrf, m->pCfg->HeadCfg.OSC.PROC_Indx, m->pCfg->HeadCfg.OSC.BtnJog_Gain * getBtnProgress());
						else
							JogProcessAndroid(intrf, m->pCfg->HeadCfg.OSC.PROC_Indx, m->pCfg->HeadCfg.OSC.BtnJog_Gain * getBtnProgress() * (-1.0));

					break;

					case BTN_JOG_MODE_DUAL_INV:

						if (!m->ToolHeadID)
							JogProcessAndroid(intrf, m->pCfg->HeadCfg.OSC.PROC_Indx, m->pCfg->HeadCfg.OSC.BtnJog_Gain * getBtnProgress());
						else
							JogProcessAndroid(intrf, m->pCfg->HeadCfg.OSC.PROC_Indx, m->pCfg->HeadCfg.OSC.BtnJog_Gain * getBtnProgress() * (-1.0));

					break;
				}

			}

		break;

		case ANDR_BTN_OSC_AMPL_POS:

			if (Process[m->pCfg->HeadCfg.OSC.PROC_Indx].Status == prcsSTATUS_Run)
			{

				strcpy(hmi->ActiveBanner, "ANDR_BTN_OSC_AMPL_POS");

				if (!intrf->_intr._GlblBtnCmd[0])
					IncrParam(curCfg, parOSC_Amplit, m->curSegm[ZONE], 1.0);

				Check_parOSC_Amplit(curCfg, hmi, m->curSegm[0]);
			}
			else if ((Process[m->pCfg->HeadCfg.OSC.PROC_Indx].Status == prcsSTATUS_Stopped) ||
			(Process[m->pCfg->HeadCfg.OSC.PROC_Indx].Status == prcsSTATUS_DirectCntrl))
			{
				strcpy(hmi->ActiveBanner, "OSC JOG RIGHT");

				switch (m->pCfg->HeadCfg.OSC.BtnJog_Mode)
				{
					case BTN_JOG_MODE_SINGLE:

						JogProcessAndroid(intrf, m->pCfg->HeadCfg.OSC.PROC_Indx,
						m->pCfg->HeadCfg.OSC.BtnJog_Gain * getBtnProgress ());

					break;

					case BTN_JOG_MODE_DUAL:

						if (m->ToolHeadID)
							JogProcessAndroid(intrf, m->pCfg->HeadCfg.OSC.PROC_Indx, m->pCfg->HeadCfg.OSC.BtnJog_Gain * getBtnProgress() * (-1.0));
						else
							JogProcessAndroid(intrf, m->pCfg->HeadCfg.OSC.PROC_Indx, m->pCfg->HeadCfg.OSC.BtnJog_Gain * getBtnProgress());

					break;

					case BTN_JOG_MODE_DUAL_INV:

						if (!m->ToolHeadID)
							JogProcessAndroid(intrf, m->pCfg->HeadCfg.OSC.PROC_Indx, m->pCfg->HeadCfg.OSC.BtnJog_Gain * getBtnProgress() * (-1.0));
						else
							JogProcessAndroid(intrf, m->pCfg->HeadCfg.OSC.PROC_Indx, m->pCfg->HeadCfg.OSC.BtnJog_Gain * getBtnProgress());

					break;
				}

			}

		break;

		case ANDR_BTN_AVC_LOCK:

			strcpy(hmi->ActiveBanner, "AVC LOCK ON / OFF");

			if (curCfg->Param_ENUM[parENUM_AVC_Mode].val[0] != 2)
			{ // AVC Mode NOT Lock

				if (!intrf->_intr._GlblBtnCmd[0])
				{

					Process[m->pCfg->HeadCfg.AVC.PROC_Indx].Param[0] =	!Process[m->pCfg->HeadCfg.AVC.PROC_Indx].Param[0]; // AVC Hold

				}

			}

		break;

		case ANDR_BTN_WIRE_DISABLE:

			strcpy(hmi->ActiveBanner, "WIRE ON/OFF");

			if (!intrf->_intr._GlblBtnCmd[0])
			{
				if (m->WireDisabled != 0)
					m->WireDisabled = 0;
				else
					m->WireDisabled = 1;

				LogTxt(&LogMgr, "Wire Disable Event %d" , (DINT)m->WireDisabled);
			}

		break;

		case ANDR_BTN_STOP:

			for (i = 0; i < PROCESS_NUM; i++)
				Process[i].fParam[0] = 0.0;

			TVL_Latch_Latched = 0;
			_TVL_Latch_Latched = TVL_Latch_Latched;
			TVL_Latch_Cnt = 0;

		break;

		default:

			for (i = 0; i < PROCESS_NUM; i++)
			{
				if (i != m->pCfg->HeadCfg.OSC.PROC_Indx)
					Process[i].fParam[0] = 0.0;
			}

			_TVL_Latch_Latched = TVL_Latch_Latched;
			TVL_Latch_Cnt = 0;
		break;
	}

	if (! (intrf->GlblBtnCmd[0] & (ANDR_BTN_OSC_AMPL_NEG + ANDR_BTN_OSC_AMPL_POS)))
		Process[m->pCfg->HeadCfg.OSC.PROC_Indx].fParam[0] = 0.0;

	if((curCalib->GenSetup[SETUP_HEAD_SETUP] == BPV_v2_MT_BO_TOS)
		|| (curCalib->GenSetup[SETUP_HEAD_SETUP] == BPV_v2_TT_BO_TOS)
		|| (curCalib->GenSetup[SETUP_HEAD_SETUP] == BPV_v2_MPGH)
		|| (curCalib->GenSetup[SETUP_HEAD_SETUP] == BPV_v2_MPGV))
		TVL_Latch_Latched = 0;

	switch (TVL_Latch_Latched)
	{
		case 1:
			JogProcessAndroid(intrf, m->pCfg->HeadCfg.TVL.PROC_Indx, -24.0);
		break;

		case 2:
			JogProcessAndroid(intrf, m->pCfg->HeadCfg.TVL.PROC_Indx, 24.0);
		break;
	}

	//	OScilation Center Jog

#ifdef MIG_PENDANT

if(intrf->WheelDelta != 0)

#else

if ((intrf->WheelDelta != 0) && (hmi->curHeadID == 0xFFFE))

#endif

	{

		if (Process[m->pCfg->HeadCfg.OSC.PROC_Indx].Status != prcsSTATUS_Init)
		{

			if ((Process[m->pCfg->HeadCfg.OSC.PROC_Indx].Status == prcsSTATUS_Stopped) ||
			(Process[m->pCfg->HeadCfg.OSC.PROC_Indx].Status == prcsSTATUS_DirectCntrl))
			{

				if (!m->pCfg->HeadCfg.OSC.WhelJog_OnlyWhenRun)
				{

					switch (m->pCfg->HeadCfg.OSC.WhelJog_Mode1)
					{
						case WHL_JOG_MODE_SINGLE:

							JogProcessAndroid(intrf, m->pCfg->HeadCfg.OSC.PROC_Indx, m->pCfg->HeadCfg.OSC.WheelJog_Gain1 * (float) intrf->WheelDelta);

						break;

						case WHL_JOG_MODE_STEP:

							Process[m->pCfg->HeadCfg.OSC.PROC_Indx].xCMD = prcsJOGpos;
							Process[m->pCfg->HeadCfg.OSC.PROC_Indx].fParam[0] = (float)intrf->WheelDelta * m->pCfg->HeadCfg.OSC.WheelJog_Gain1;

						break;

						case WHL_JOG_MODE_DUAL:

							if (m->ToolHeadID)
								JogProcessAndroid(intrf, m->pCfg->HeadCfg.OSC.PROC_Indx, m->pCfg->HeadCfg.OSC.WheelJog_Gain1 * (float) intrf->WheelDelta);
							else
								JogProcessAndroid(intrf, m->pCfg->HeadCfg.OSC.PROC_Indx, m->pCfg->HeadCfg.OSC.WheelJog_Gain1 * (float) intrf->WheelDelta * (-1.0));

						break;

						case WHL_JOG_MODE_DUAL_INV:

							if (m->ToolHeadID)
								JogProcessAndroid(intrf, m->pCfg->HeadCfg.OSC.PROC_Indx, m->pCfg->HeadCfg.OSC.WheelJog_Gain1 * (float) intrf->WheelDelta);
							else
								JogProcessAndroid(intrf, m->pCfg->HeadCfg.OSC.PROC_Indx, m->pCfg->HeadCfg.OSC.WheelJog_Gain1 * (float) intrf->WheelDelta * (-1.0));

						break;
					}
				}

			}
			else
			{

				Process[m->pCfg->HeadCfg.OSC.PROC_Indx].xCMD = prcsJOGpos;

				switch (m->pCfg->HeadCfg.OSC.WhelJog_Mode2)
				{
					case WHL_JOG_MODE_SINGLE:
					case WHL_JOG_MODE_STEP:

						Process[m->pCfg->HeadCfg.OSC.PROC_Indx].fParam[0] = (float)intrf->WheelDelta * m->pCfg->HeadCfg.OSC.WheelJog_Gain2;

					break;

					case WHL_JOG_MODE_DUAL:

						if (m->ToolHeadID)
							Process[m->pCfg->HeadCfg.OSC.PROC_Indx].fParam[0] = (float)intrf->WheelDelta * m->pCfg->HeadCfg.OSC.WheelJog_Gain2;
						else
							Process[m->pCfg->HeadCfg.OSC.PROC_Indx].fParam[0] = (float)intrf->WheelDelta * m->pCfg->HeadCfg.OSC.WheelJog_Gain2 * (-1.0);

					break;

					case WHL_JOG_MODE_DUAL_INV:

						if (!m->ToolHeadID)
							Process[m->pCfg->HeadCfg.OSC.PROC_Indx].fParam[0] = (float)intrf->WheelDelta * m->pCfg->HeadCfg.OSC.WheelJog_Gain2;
						else
							Process[m->pCfg->HeadCfg.OSC.PROC_Indx].fParam[0] = (float)intrf->WheelDelta * m->pCfg->HeadCfg.OSC.WheelJog_Gain2 * (-1.0);

					break;
				}

			}

		}
	}

}

void StopCalibrationModeAndroidButtons(MASTER_typ * m, HMI_typ * hmi, HMI_INTRF_typ * intrf, LCD_MGR_obj * lcd)
{

	StopModeAndroidButtons(m, hmi, intrf, lcd);

	return;

}

void RunModeAndroidButtons(MASTER_typ * m, HMI_typ * hmi, HMI_INTRF_typ * intrf, LCD_MGR_obj * lcd)
{
UINT			i;
UINT			par;
CurCfg_typ *	curCfg;
curCfg				= m->pCurCfg;

	if (!curCfg)
		return;

 //if((Weld_Report_Status != 1) ||  ((curCalib->GenSetup[SETUP_EXTRAS]&0x1) == 0)){
 if(((curCalib->GenSetup[SETUP_EXTRAS]&0x1) == 0)){

	switch (intrf->GlblBtnCmd[0])
	{
		case ANDR_BTN_ARC_AMPS_NEG:

			if (m->AndIntrf[0].GlblBtnLED[1] &0x2){

				strcpy(hmi->ActiveBanner, "WB#1 JOG REV");
				JogProcessAndroid(intrf, m->pCfg->HeadCfg.WB[WB_UD].PROC_Indx,(-1.0));

			}else{

				strcpy(hmi->ActiveBanner, " ARC AMPS minus ");

				if (!intrf->_intr._GlblBtnCmd[0])
					ChangeParam(parTIG_AmpSP , -1 );
			}

		break;

		case ANDR_BTN_ARC_AMPS_POS:

			if (m->AndIntrf[0].GlblBtnLED[1] &0x2){

				strcpy(hmi->ActiveBanner, "WB#1 JOG FWD");
				JogProcessAndroid(intrf, m->pCfg->HeadCfg.WB[WB_UD].PROC_Indx,(1.0));

			}else{

				strcpy(hmi->ActiveBanner, " ARC AMPS plus ");

				if (!intrf->_intr._GlblBtnCmd[0])
					ChangeParam(parTIG_AmpSP , 1 );
			}

		break;

		case ANDR_BTN_TRAVEL_SPEED_NEG:

			if (m->AndIntrf[0].GlblBtnLED[1] &0x2){

				strcpy(hmi->ActiveBanner, "WB#2 JOG REV");
				JogProcessAndroid(intrf, m->pCfg->HeadCfg.WB[WB_LR].PROC_Indx,(-1.0));

			}else{

				strcpy(hmi->ActiveBanner, " TRAVEL SPEED minus ");

				if (!intrf->_intr._GlblBtnCmd[0])
					ChangeParam(parTVL_VelSP , -1 );

			}

		break;

		case ANDR_BTN_TRAVEL_SPEED_POS:

			if (m->AndIntrf[0].GlblBtnLED[1] &0x2){

				strcpy(hmi->ActiveBanner, "WB#2 JOG FWD");
				JogProcessAndroid(intrf, m->pCfg->HeadCfg.WB[WB_LR].PROC_Indx,(1.0));

			}else{

				strcpy(hmi->ActiveBanner, " TRAVEL SPEED plus");

				if (!intrf->_intr._GlblBtnCmd[0])
					ChangeParam(parTVL_VelSP , 1 );

			}

		break;

		case ANDR_BTN_WIRE_SPEED_NEG:

			if (m->AndIntrf[0].GlblBtnLED[1] &0x2){

				Hardware[1].Outp[9] = 1; // Lights OFF (NC) on camera

			}else{

				strcpy(hmi->ActiveBanner, "WIRE SPEED minus");

				if (!intrf->_intr._GlblBtnCmd[0])
					ChangeParam(parWF_SpeedSP , -1 );

			}

		break;

		case ANDR_BTN_WIRE_SPEED_POS:

			if (m->AndIntrf[0].GlblBtnLED[1] &0x2){

				Hardware[1].Outp[9] = 0; // Lights ON (NC) on camera

			}else{

				strcpy(hmi->ActiveBanner, "WIRE SPEED plus");

				if(!intrf->_intr._GlblBtnCmd[0])
					ChangeParam(parWF_SpeedSP , 1 );

			}

		break;

		case ANDR_BTN_AVC_VOLTS_NEG:

			if(Process[m->pCfg->HeadCfg.AVC.PROC_Indx].Status == prcsSTATUS_AVC_Hold )
				Process[m->pCfg->HeadCfg.AVC.PROC_Indx].fParam[0] = m->pCfg->HeadCfg.AVC.BtnJog_Gain * getBtnProgress() * (-1.0);

			else if (m->TestMode){

				strcpy(hmi->ActiveBanner, " AVC JOG DOWN ");
				JogProcessAndroid(intrf, m->pCfg->HeadCfg.AVC.PROC_Indx, m->pCfg->HeadCfg.AVC.BtnJog_Gain * getBtnProgress() * (-1.0));

			}
			else{

				strcpy(hmi->ActiveBanner, "AVC VOLT minus");

				if (!intrf->_intr._GlblBtnCmd[0])
					ChangeParam(parAVC_VoltSP , -1 );

			}

		break;

		case ANDR_BTN_AVC_VOLTS_POS:

			if(Process[m->pCfg->HeadCfg.AVC.PROC_Indx].Status == prcsSTATUS_AVC_Hold )
				Process[m->pCfg->HeadCfg.AVC.PROC_Indx].fParam[0] = m->pCfg->HeadCfg.AVC.BtnJog_Gain * getBtnProgress();

			else if (m->TestMode){

				strcpy(hmi->ActiveBanner, " AVC JOG UP ");
				JogProcessAndroid(intrf, m->pCfg->HeadCfg.AVC.PROC_Indx, m->pCfg->HeadCfg.AVC.BtnJog_Gain * getBtnProgress());

			}
			else{

				strcpy(hmi->ActiveBanner, "AVC VOLT plus");

				if (!intrf->_intr._GlblBtnCmd[0])
					ChangeParam(parAVC_VoltSP , 1 );

			}

		break;

		case ANDR_BTN_OSC_SPEED_NEG:
			strcpy(hmi->ActiveBanner, "OSC	TIME minus");

			if(m->pCfg->HeadCfg.OSC.DwellDir){

				if (m->AndIntrf[0].GlblBtnLED[1] &0x2){

					par = parOSC_Dwell_Out;
				}
				else if (m->AndIntrf[0].GlblBtnLED[1] &0x1){

					par = parOSC_Dwell_In;
				}
				else
					par = parOSC_Excur;

			}
			else{

				if (m->AndIntrf[0].GlblBtnLED[1] &0x1){

					par = parOSC_Dwell_In;
				}
				else if (m->AndIntrf[0].GlblBtnLED[1] &0x2){

					par = parOSC_Dwell_Out;
				}
				else
					par = parOSC_Excur;

			}

			if (!intrf->_intr._GlblBtnCmd[0])
			{
				DecrParam(curCfg, par, m->curSegm[ZONE], 1.0);

				if (par == parOSC_Excur)
					Check_parOSC_Excur(curCfg, hmi, m->curSegm[ZONE]);

				if (! (curCalib->GenSetup[SETUP_WHERE_FILL] == 2)) //Not only Editor
					Fill_Segments(curCfg, par, m->curSegm[ZONE], curCalib->GenSetup[SETUP_AUTO_FILL], m->sm.Step);

			}

		break;

		case ANDR_BTN_OSC_SPEED_POS:
			strcpy(hmi->ActiveBanner, "OSC	TIME plus");

			if(m->pCfg->HeadCfg.OSC.DwellDir){

				if (m->AndIntrf[0].GlblBtnLED[1] &0x2){

					par = parOSC_Dwell_Out;
				}
				else if (m->AndIntrf[0].GlblBtnLED[1] &0x1){

					par = parOSC_Dwell_In;
				}
				else
					par = parOSC_Excur;

			}
			else{

				if (m->AndIntrf[0].GlblBtnLED[1] &0x1){

					par = parOSC_Dwell_In;
				}
				else if (m->AndIntrf[0].GlblBtnLED[1] &0x2){

					par = parOSC_Dwell_Out;
				}
				else
					par = parOSC_Excur;

			}

			if (!intrf->_intr._GlblBtnCmd[0])
			{
				IncrParam(curCfg, par, m->curSegm[ZONE], 1.0);

				if (par == parOSC_Excur)
					Check_parOSC_Excur(curCfg, hmi, m->curSegm[ZONE]);

				if (! (curCalib->GenSetup[SETUP_WHERE_FILL] == 2)) //Not only Editor
					Fill_Segments(curCfg, par, m->curSegm[ZONE], curCalib->GenSetup[SETUP_AUTO_FILL], m->sm.Step);

			}

		break;

		case ANDR_BTN_OSC_AMPL_NEG:
			strcpy(hmi->ActiveBanner, "OSC AMPLITUDE minus");

			if (!intrf->_intr._GlblBtnCmd[0])
			{
				DecrParam(curCfg, parOSC_Amplit, m->curSegm[ZONE], 1.0);

				Check_parOSC_Amplit(curCfg, hmi, m->curSegm[ZONE]);

				if (! (curCalib->GenSetup[SETUP_WHERE_FILL] == 2)) //Not only Editor
					Fill_Segments(curCfg, parOSC_Amplit, m->curSegm[ZONE], curCalib->GenSetup[SETUP_AUTO_FILL], m->sm.Step);

			}

		break;

		case ANDR_BTN_OSC_AMPL_POS:
			strcpy(hmi->ActiveBanner, "OSC AMPLITUDE plus");

			if (!intrf->_intr._GlblBtnCmd[0])
			{
				IncrParam(curCfg, parOSC_Amplit, m->curSegm[ZONE], 1.0);

				Check_parOSC_Amplit(curCfg, hmi, m->curSegm[ZONE]);

			if (! (curCalib->GenSetup[SETUP_WHERE_FILL] == 2)) //Not only Editor
				Fill_Segments(curCfg, parOSC_Amplit, m->curSegm[ZONE], curCalib->GenSetup[SETUP_AUTO_FILL],	m->sm.Step);

			}

		break;

		case ANDR_BTN_AVC_LOCK:
			strcpy(hmi->ActiveBanner, "AVC LOCK ON / OFF");

			if (curCfg->Param_ENUM[parENUM_AVC_Mode].val[0] != 2)
			{ // AVC Mode NOT Lock

				if (!intrf->_intr._GlblBtnCmd[0])
				{

					Process[m->pCfg->HeadCfg.AVC.PROC_Indx].Param[0] =	!Process[m->pCfg->HeadCfg.AVC.PROC_Indx].Param[0]; // AVC Hold

				}

			}

		break;

		case ANDR_BTN_WIRE_DISABLE:
			strcpy(hmi->ActiveBanner, "WIRE ON/OFF");

			if (!intrf->_intr._GlblBtnCmd[0])
			{

				if (m->WireDisabled != 0)
					m->WireDisabled = 0;
				else
					m->WireDisabled = 1;

				LogTxt(&LogMgr, "Wire Disable Event %d" , (DINT)m->WireDisabled);
			}

		break;

		default:

			for (i = 0; i < PROCESS_NUM; i++)
			Process[i].fParam[0] = 0.0;

		break;
	}

}
 else{

	switch (intrf->GlblBtnCmd[0])
	{
		case ANDR_BTN_WIRE_DISABLE:
			strcpy(hmi->ActiveBanner, "WIRE ON/OFF");

			if (!intrf->_intr._GlblBtnCmd[0])
			{

				if (m->WireDisabled != 0)
					m->WireDisabled = 0;
				else
					m->WireDisabled = 1;

				LogTxt(&LogMgr, "Wire Disable Event %d" , (DINT)m->WireDisabled);
			}

		break;

		default:

			for (i = 0; i < PROCESS_NUM; i++)
			Process[i].fParam[0] = 0.0;

		break;

	}

 }

//	OScilation Center Jog
#ifdef MIG_PENDANT

if(intrf->WheelDelta != 0)

#else

if ((intrf->WheelDelta != 0) && (hmi->curHeadID == 0xFFFE))

#endif
{

// only jog on Run and Alternate Run screen

	if (Process[m->pCfg->HeadCfg.OSC.PROC_Indx].Status != prcsSTATUS_Init)
	{

		if ((Process[m->pCfg->HeadCfg.OSC.PROC_Indx].Status == prcsSTATUS_Stopped) ||
		(Process[m->pCfg->HeadCfg.OSC.PROC_Indx].Status == prcsSTATUS_DirectCntrl))
		{

			switch (m->pCfg->HeadCfg.OSC.WhelJog_Mode1)
			{
				case WHL_JOG_MODE_SINGLE:

					JogProcessAndroid(intrf, m->pCfg->HeadCfg.OSC.PROC_Indx,
					m->pCfg->HeadCfg.OSC.WheelJog_Gain1 * (float) intrf->WheelDelta);

				break;

				case WHL_JOG_MODE_STEP:

					Process[m->pCfg->HeadCfg.OSC.PROC_Indx].xCMD = prcsJOGpos;
					Process[m->pCfg->HeadCfg.OSC.PROC_Indx].fParam[0] = (float)
					intrf->WheelDelta * m->pCfg->HeadCfg.OSC.WheelJog_Gain1;

				break;

				case WHL_JOG_MODE_DUAL:

					if (m->ToolHeadID)
						JogProcessAndroid(intrf, m->pCfg->HeadCfg.OSC.PROC_Indx,m->pCfg->HeadCfg.OSC.WheelJog_Gain1 * (float) intrf->WheelDelta);
					else
						JogProcessAndroid(intrf, m->pCfg->HeadCfg.OSC.PROC_Indx,m->pCfg->HeadCfg.OSC.WheelJog_Gain1 * (float) intrf->WheelDelta * (-1.0));

				break;

				case WHL_JOG_MODE_DUAL_INV:

					if (m->ToolHeadID)
						JogProcessAndroid(intrf, m->pCfg->HeadCfg.OSC.PROC_Indx,m->pCfg->HeadCfg.OSC.WheelJog_Gain1 * (float) intrf->WheelDelta);
					else
						JogProcessAndroid(intrf, m->pCfg->HeadCfg.OSC.PROC_Indx,m->pCfg->HeadCfg.OSC.WheelJog_Gain1 * (float) intrf->WheelDelta * (-1.0));

				break;
				}

		}
		else
		{

			Process[m->pCfg->HeadCfg.OSC.PROC_Indx].xCMD = prcsJOGpos;

			switch (m->pCfg->HeadCfg.OSC.WhelJog_Mode2)
			{
				case WHL_JOG_MODE_SINGLE:
				case WHL_JOG_MODE_STEP:

					Process[m->pCfg->HeadCfg.OSC.PROC_Indx].fParam[0] = (float)intrf->WheelDelta * m->pCfg->HeadCfg.OSC.WheelJog_Gain2;
				break;

				case WHL_JOG_MODE_DUAL:

					if (m->ToolHeadID)
						Process[m->pCfg->HeadCfg.OSC.PROC_Indx].fParam[0] = (float)intrf->WheelDelta * m->pCfg->HeadCfg.OSC.WheelJog_Gain2;
					else
						Process[m->pCfg->HeadCfg.OSC.PROC_Indx].fParam[0] = (float)intrf->WheelDelta * m->pCfg->HeadCfg.OSC.WheelJog_Gain2 * (-1.0);

				break;

				case WHL_JOG_MODE_DUAL_INV:

					if (!m->ToolHeadID)
						Process[m->pCfg->HeadCfg.OSC.PROC_Indx].fParam[0] = (float)intrf->WheelDelta * m->pCfg->HeadCfg.OSC.WheelJog_Gain2;
					else
						Process[m->pCfg->HeadCfg.OSC.PROC_Indx].fParam[0] = (float)intrf->WheelDelta * m->pCfg->HeadCfg.OSC.WheelJog_Gain2 * (-1.0);

				break;
				}

			}

		}
	}

}

void RunCalibrationModeAndroidButtons(MASTER_typ * m, HMI_typ * hmi, HMI_INTRF_typ * intrf, LCD_MGR_obj * lcd)
{
	StopModeAndroidButtons(m, hmi, intrf, lcd);
	return;
}

DINT CalibrationSequence(MASTER_typ * m, HMI_typ * hmi, plcbit StartBtn, plcbit StopBtn)
{
UINT			i, status;
DINT			ret;

//Cfg_typ *cfg;
CurCfg_typ *	curCfg;
CurCalib_typ *	curCalib, *defCalib;

	//Scaled_Var_obj *var;
	//cfg = (Cfg_typ*) m->pCfg;
	curCfg	= (CurCfg_typ *)m->pCurCfg;
	curCalib = (CurCalib_typ *)	m->pCalib;
	defCalib = (CurCalib_typ *)	m->pDefaultCalib;

	//var = (Scaled_Var_obj*) m->pScaledVar;
	///////////////////////////////
	// Button Start and Stop
	ret = 1; // Stop

	switch (m->CalibType)
	{
	case CALIB_TVL:

		if ((Process[m->pCfg->HeadCfg.TVL.PROC_Indx].Status == prcsSTATUS_Stopped) ||
		(Process[m->pCfg->HeadCfg.TVL.PROC_Indx].Status == prcsSTATUS_DirectCntrl))
		{

			if (StartBtn)
				Process[m->pCfg->HeadCfg.TVL.PROC_Indx].xCMD = prcsCalib;

		}

		if(StopBtn)
			CalibrTMR.IN = 0;

		else if (StartBtn){

			if(Process[m->pCfg->HeadCfg.TVL.PROC_Indx].Status == prcsSTATUS_ForceCalib){

				if(!CalibrTMR.IN)
					TimerStart(&CalibrTMR, 600.0);

			}

		}

		switch (hmi->CalibStep)
		{

			case 1:
			case 2: // Low Vel

				//if(StartBtn || KK_Functionality){
				if (Process[m->pCfg->HeadCfg.TVL.PROC_Indx].Param[1] &0x2)
				{

					Process[m->pCfg->HeadCfg.TVL.PROC_Indx].fParam[1] =	getFromCalib(curCfg->Param[parTVL_CalibVel1].val[0], &curCalib->Points[CALIB_TVL_SPEED_CMD], CALIB_2POINTS);
					hmi->CalibPoint[hmi->CalibStep] = 0;
					hmi->CalibPointCmd[hmi->CalibStep] = Process[m->pCfg->HeadCfg.TVL.PROC_Indx].fParam[1];

				}
				else
				{

					Process[m->pCfg->HeadCfg.TVL.PROC_Indx].fParam[1] =	getFromCalib(curCfg->Param[parTVL_CalibVel1].val[0], &curCalib->Points[CALIB_TVL_SPEED_CMD], CALIB_2POINTS_4OFF);
					hmi->CalibPoint[hmi->CalibStep] = 4;
					hmi->CalibPointCmd[hmi->CalibStep] = Process[m->pCfg->HeadCfg.TVL.PROC_Indx].fParam[1];

				}

				//}
				if (KK_ManualCalib)
					Process[m->pCfg->HeadCfg.TVL.PROC_Indx].fParam[1] = KK_ManualCalib_set_value;

			break;

			case 3:
			case 4:

				// High Vel
				//if(StartBtn || KK_Functionality){
				if (Process[m->pCfg->HeadCfg.TVL.PROC_Indx].Param[1] &0x2)
				{

					Process[m->pCfg->HeadCfg.TVL.PROC_Indx].fParam[1] =	getFromCalib(curCfg->Param[parTVL_CalibVel2].val[0], &curCalib->Points[CALIB_TVL_SPEED_CMD], CALIB_2POINTS);
					hmi->CalibPoint[hmi->CalibStep] = 2;
					hmi->CalibPointCmd[hmi->CalibStep] = Process[m->pCfg->HeadCfg.TVL.PROC_Indx].fParam[1];

				}
				else
				{
					Process[m->pCfg->HeadCfg.TVL.PROC_Indx].fParam[1] =	getFromCalib(curCfg->Param[parTVL_CalibVel2].val[0], &curCalib->Points[CALIB_TVL_SPEED_CMD], CALIB_2POINTS_4OFF);
					hmi->CalibPoint[hmi->CalibStep] = 6;
					hmi->CalibPointCmd[hmi->CalibStep] = Process[m->pCfg->HeadCfg.TVL.PROC_Indx].fParam[1];
				}

				//}
				if (KK_ManualCalib)
				Process[m->pCfg->HeadCfg.TVL.PROC_Indx].fParam[1] = KK_ManualCalib_set_value;

			break;

			default:
				Process[m->pCfg->HeadCfg.TVL.PROC_Indx].fParam[1] = 0.0;
			break;
		}

	break;

	///////////////////////////////////////////
	case CALIB_WF:

		if((Process[m->pCfg->HeadCfg.WF.PROC_Indx].Status == prcsSTATUS_Stopped) ||
		(Process[m->pCfg->HeadCfg.WF.PROC_Indx].Status == prcsSTATUS_DirectCntrl))
		{
			if (StartBtn)
				Process[m->pCfg->HeadCfg.WF.PROC_Indx].xCMD = prcsCalib;
		}

		if(TimerIsTimeOut(&CalibrTMR))
		{
			CalibrTMR.IN = 0;
			CalibrTMR.Q = 0;
			Process[m->pCfg->HeadCfg.WF.PROC_Indx].xCMD = prcsHalt;
		}

		switch (hmi->CalibStep)
		{

			case 1:
			case 3: // Low Vel

				if (StartBtn)
					TimerStart(&CalibrTMR, curCfg->Param[parGEN_CalibTime1].val[0]);

				//if(StartBtn || KK_Functionality){
				if (Process[m->pCfg->HeadCfg.WF.PROC_Indx].Param[1])
				{
					hmi->CalibPoint[hmi->CalibStep] = 0;
					Process[m->pCfg->HeadCfg.WF.PROC_Indx].fParam[1] = getFromCalib(curCfg->Param[parWF_CalibVel1].val[0], &curCalib->Points[CALIB_WF_SPEED_CMD], CALIB_2POINTS);
					hmi->CalibPointCmd[hmi->CalibStep] = Process[m->pCfg->HeadCfg.WF.PROC_Indx].fParam[1];
				}
				else
				{
					hmi->CalibPoint[hmi->CalibStep] = 4;
					Process[m->pCfg->HeadCfg.WF.PROC_Indx].fParam[1] = getFromCalib(curCfg->Param[parWF_CalibVel1].val[0], &curCalib->Points[CALIB_WF_SPEED_CMD], CALIB_2POINTS_4OFF);
					hmi->CalibPointCmd[hmi->CalibStep] = Process[m->pCfg->HeadCfg.WF.PROC_Indx].fParam[1];
				}

				//}
				if (KK_ManualCalib)
					Process[m->pCfg->HeadCfg.WF.PROC_Indx].fParam[1] = KK_ManualCalib_set_value;

			break;

			case 2:
			case 4: // High Vel

				if (StartBtn)
					TimerStart(&CalibrTMR, curCfg->Param[parGEN_CalibTime2].val[0]);

				//if(StartBtn || KK_Functionality){
				if (Process[m->pCfg->HeadCfg.WF.PROC_Indx].Param[1])
				{
					hmi->CalibPoint[hmi->CalibStep] = 2;
					Process[m->pCfg->HeadCfg.WF.PROC_Indx].fParam[1] = getFromCalib(curCfg->Param[parWF_CalibVel2].val[0], &curCalib->Points[CALIB_WF_SPEED_CMD], CALIB_2POINTS);
					hmi->CalibPointCmd[hmi->CalibStep] = Process[m->pCfg->HeadCfg.WF.PROC_Indx].fParam[1];
				}
				else
				{
					hmi->CalibPoint[hmi->CalibStep] = 6;
					Process[m->pCfg->HeadCfg.WF.PROC_Indx].fParam[1] = getFromCalib(curCfg->Param[parWF_CalibVel2].val[0], &curCalib->Points[CALIB_WF_SPEED_CMD], CALIB_2POINTS_4OFF);
					hmi->CalibPointCmd[hmi->CalibStep] = Process[m->pCfg->HeadCfg.WF.PROC_Indx].fParam[1];
				}

				//}
				if (KK_ManualCalib)
					Process[m->pCfg->HeadCfg.WF.PROC_Indx].fParam[1] = KK_ManualCalib_set_value;

			break;

			default:

				Process[m->pCfg->HeadCfg.WF.PROC_Indx].fParam[1] = 0.0;

			break;
		}

	break;

	//////////////////////////////////////////////////////////////////
	case CALIB_TIG_PS:

		if ((Process[m->pCfg->HeadCfg.TIG.PROC_Indx].Status == prcsSTATUS_Stopped) ||
		(Process[m->pCfg->HeadCfg.TIG.PROC_Indx].Status == prcsSTATUS_DirectCntrl))
		{
			if (StartBtn){

				switch(curCfg->Param_ENUM[parENUM_TIG_Cal_Mode].val[0]){

					case 1: // Load Bank

						Process[m->pCfg->HeadCfg.TIG.PROC_Indx].xCMD = prcsCalib;

					break;

					default: // Arc start

						if(AmpsCalib_step == 0)
							AmpsCalib_step = 1;

					break;

				}

			}
		}

		switch(AmpsCalib_step){

			 case 0:

			 break;

			 case 1:

			 	if (ErrorMgr.Error){
					 AmpsCalib_step = 100;
					 break;

			 	}

				else if(StopBtn){

					AmpsCalib_step = 10;
					break;
				}

			 	if (!m->TestMode)
				{
					Process[m->pCfg->HeadCfg.GAS.PROC_Indx].xCMD = prcsSTART;
					Process[m->pCfg->HeadCfg.COOL.PROC_Indx].xCMD = prcsSTART;
				}

				if(m->TestMode)
				{

					Process[m->pCfg->HeadCfg.AVC.PROC_Indx].TestMode = 1;
					Process[m->pCfg->HeadCfg.TIG.PROC_Indx].xCMD = prcsHalt;

				}
				else
				{

					if ((Process[m->pCfg->HeadCfg.GAS.PROC_Indx].Status == prcsSTATUS_Run) &&
					(Process[m->pCfg->HeadCfg.COOL.PROC_Indx].Status == prcsSTATUS_Run))
					{
						Process[m->pCfg->HeadCfg.AVC.PROC_Indx].TestMode = 0;
						Process[m->pCfg->HeadCfg.TIG.PROC_Indx].xCMD = prcsCalib;

					}
					else
						break;

				}

				Process[m->pCfg->HeadCfg.AVC.PROC_Indx].xCMD = prcsSTART;

				AmpsCalib_step++;

			 break;

			 case 2:

				if (ErrorMgr.Error){
					 AmpsCalib_step = 100;
					 break;

			 	}

				else if(StopBtn){

					AmpsCalib_step = 10;
					break;
				}

				 if (Process[m->pCfg->HeadCfg.AVC.PROC_Indx].Status == prcsSTATUS_Run)
				 {

	 				/* AVC */
					 Process[m->pCfg->HeadCfg.OSC.PROC_Indx].xCMD = prcsSTART;
					 Process[m->pCfg->HeadCfg.OSC.PROC_Indx].Param[0] = 1; // Start without ramp

					 /*  TVL */
					 Process[m->pCfg->HeadCfg.TVL.PROC_Indx].Param[2] = 0; // No Auto stop
					 Process[m->pCfg->HeadCfg.TVL.PROC_Indx].xCMD = prcsSTART;

					AmpsCalib_step++;
				 }

			 break;

			 case 3:

			 	if (ErrorMgr.Error){

					 AmpsCalib_step = 100;

			 	}

				else if(StopBtn){

					AmpsCalib_step = 10;
				}

			 break;

			 case 10: // Stop sequence

				if (ErrorMgr.Error){
					 AmpsCalib_step = 100;
					 break;

			 	}

				Process[m->pCfg->HeadCfg.OSC.PROC_Indx].xCMD = prcsQuickSTOP;
				Process[m->pCfg->HeadCfg.GAS.PROC_Indx].xCMD = prcsSTOP;
				Process[m->pCfg->HeadCfg.AVC.PROC_Indx].xCMD = prcsHalt;

				Process[m->pCfg->HeadCfg.TIG.PROC_Indx].xCMD = prcsHalt;
				Process[m->pCfg->HeadCfg.TVL.PROC_Indx].xCMD = prcsHalt;

				AmpsCalib_step++;

			 break;

			 case 11:

			 	if (ErrorMgr.Error){
					 AmpsCalib_step = 100;
					 break;

			 	}

				else if(StopBtn){

					AmpsCalib_step = 100;
					break;
				}

				status = 1;
				if (Process[m->pCfg->HeadCfg.TVL.PROC_Indx].Status != prcsSTATUS_Stopped)
					status = 0;

				if (Process[m->pCfg->HeadCfg.OSC.PROC_Indx].Status != prcsSTATUS_Stopped)
					status = 0;

				if (Process[m->pCfg->HeadCfg.AVC.PROC_Indx].Status != prcsSTATUS_Stopped)
					status = 0;

				if (Process[m->pCfg->HeadCfg.TIG.PROC_Indx].Status != prcsSTATUS_Stopped)
					status = 0;

				//if (Process[m->pCfg->HeadCfg.GAS.PROC_Indx].Status != prcsSTATUS_Stopped)
					//status = 0;

				if(status)
					AmpsCalib_step = 0;

			 break;

			case 100:

				if (Process[m->pCfg->HeadCfg.TVL.PROC_Indx].Status != prcsSTATUS_Stopped)
				   Process[m->pCfg->HeadCfg.TVL.PROC_Indx].xCMD = prcsHalt;

				if (Process[m->pCfg->HeadCfg.OSC.PROC_Indx].Status != prcsSTATUS_Stopped)
				   Process[m->pCfg->HeadCfg.OSC.PROC_Indx].xCMD = prcsHalt;

				if (Process[m->pCfg->HeadCfg.AVC.PROC_Indx].Status != prcsSTATUS_Stopped)
				   Process[m->pCfg->HeadCfg.AVC.PROC_Indx].xCMD = prcsHalt;

				if (Process[m->pCfg->HeadCfg.TIG.PROC_Indx].Status != prcsSTATUS_Stopped)
				   Process[m->pCfg->HeadCfg.TIG.PROC_Indx].xCMD = prcsHalt;

				if (Process[m->pCfg->HeadCfg.GAS.PROC_Indx].Status != prcsSTATUS_Stopped)
				   Process[m->pCfg->HeadCfg.GAS.PROC_Indx].xCMD = prcsSTOP;

				AmpsCalib_step = 0;

			break;

			default:

				AmpsCalib_step = 0;

			break;

		}

		switch (hmi->CalibStep)
		{
			case 1:
				//if(StartBtn || KK_Functionality){
				hmi->CalibPoint[hmi->CalibStep] = 0;
				Process[m->pCfg->HeadCfg.TIG.PROC_Indx].fParam[1] =	getFromCalib(curCfg->Param[parTIG_CalibAmp1].val[0], &curCalib->Points[CALIB_TIG_AMPS_CMD],	CALIB_2POINTS);
				hmi->CalibPointCmd[hmi->CalibStep] = Process[m->pCfg->HeadCfg.TIG.PROC_Indx].fParam[1];

				//}
				if(KK_ManualCalib)
					Process[m->pCfg->HeadCfg.TIG.PROC_Indx].fParam[1] = KK_ManualCalib_set_value;

			break;

			case 2:
				//if(StartBtn || KK_Functionality){
				hmi->CalibPoint[hmi->CalibStep] = 2;
				Process[m->pCfg->HeadCfg.TIG.PROC_Indx].fParam[1] =	getFromCalib(curCfg->Param[parTIG_CalibAmp2].val[0], &curCalib->Points[CALIB_TIG_AMPS_CMD],	CALIB_2POINTS);
				hmi->CalibPointCmd[hmi->CalibStep] = Process[m->pCfg->HeadCfg.TIG.PROC_Indx].fParam[1];

				//}
				if (KK_ManualCalib)
					Process[m->pCfg->HeadCfg.TIG.PROC_Indx].fParam[1] = KK_ManualCalib_set_value;

			break;

			default:

				Process[m->pCfg->HeadCfg.TIG.PROC_Indx].fParam[1] = 0.0;

			break;
		}

	break;

	//////////////////////////////////////////////////////////////////
	case CALIB_HW_PS:
		if ((Process[m->pCfg->HeadCfg.HW.PROC_Indx].Status == prcsSTATUS_Stopped) ||
		(Process[m->pCfg->HeadCfg.HW.PROC_Indx].Status == prcsSTATUS_DirectCntrl))
		{
			if (StartBtn)
				Process[m->pCfg->HeadCfg.HW.PROC_Indx].xCMD = prcsCalib;
		}

		switch (hmi->CalibStep)
		{
			case 1:
				//if(StartBtn || KK_Functionality){
				hmi->CalibPoint[hmi->CalibStep] = 0;
				Process[m->pCfg->HeadCfg.HW.PROC_Indx].fParam[1] = getFromCalib(curCfg->Param[parHW_CalibAmp1].val[0], &curCalib->Points[CALIB_HW_AMPS_CMD], CALIB_2POINTS);
				hmi->CalibPointCmd[hmi->CalibStep] = Process[m->pCfg->HeadCfg.HW.PROC_Indx].fParam[1];

				//}
				if (KK_ManualCalib)
					Process[m->pCfg->HeadCfg.HW.PROC_Indx].fParam[1] = KK_ManualCalib_set_value;

			break;

			case 2:
				//if(StartBtn || KK_Functionality){
				hmi->CalibPoint[hmi->CalibStep] = 2;
				Process[m->pCfg->HeadCfg.HW.PROC_Indx].fParam[1] = getFromCalib(curCfg->Param[parHW_CalibAmp2].val[0], &curCalib->Points[CALIB_HW_AMPS_CMD], CALIB_2POINTS);
				hmi->CalibPointCmd[hmi->CalibStep] = Process[m->pCfg->HeadCfg.HW.PROC_Indx].fParam[1];

				//}
				if (KK_ManualCalib)
					Process[m->pCfg->HeadCfg.HW.PROC_Indx].fParam[1] = KK_ManualCalib_set_value;

			break;

			default:

				Process[m->pCfg->HeadCfg.HW.PROC_Indx].fParam[1] = 0.0;

			break;
		}

	break;

	///////////////////////////////////////////
	}

	status = 1;

	if (Process[m->pCfg->HeadCfg.TVL.PROC_Indx].Status != prcsSTATUS_Stopped)
		status = 0;

	if (Process[m->pCfg->HeadCfg.OSC.PROC_Indx].Status != prcsSTATUS_Stopped)
		status = 0;

	if (Process[m->pCfg->HeadCfg.AVC.PROC_Indx].Status != prcsSTATUS_Stopped)
		status = 0;

	if (Process[m->pCfg->HeadCfg.WF.PROC_Indx].Status != prcsSTATUS_Stopped)
		status = 0;

	if (Process[m->pCfg->HeadCfg.WP.PROC_Indx].Status != prcsSTATUS_Stopped)
		status = 0;

	if (Process[m->pCfg->HeadCfg.TIG.PROC_Indx].Status != prcsSTATUS_Stopped)
		status = 0;

	if (Process[m->pCfg->HeadCfg.HW.PROC_Indx].Status != prcsSTATUS_Stopped)
		status = 0;

	if (Process[m->pCfg->HeadCfg.GAS.PROC_Indx].Status != prcsSTATUS_Stopped)
		status = 0;

		//intrf->GlblBtnLED[0] += BTN_B0; //SEQ_STOP_LED
		if (StopBtn)
		{ // Stop Button

			if (!status)
			{

				if(AmpsCalib_step == 0){ // No TIG calibration in ARC mode

					Process[m->pCfg->HeadCfg.TVL.PROC_Indx].xCMD = prcsHalt;
					Process[m->pCfg->HeadCfg.OSC.PROC_Indx].xCMD = prcsHalt;
					Process[m->pCfg->HeadCfg.AVC.PROC_Indx].xCMD = prcsHalt;
					Process[m->pCfg->HeadCfg.WF.PROC_Indx].xCMD = prcsHalt;
					Process[m->pCfg->HeadCfg.GAS.PROC_Indx].xCMD = prcsHalt;
					Process[m->pCfg->HeadCfg.WP.PROC_Indx].xCMD = prcsHalt;
					Process[m->pCfg->HeadCfg.TIG.PROC_Indx].xCMD = prcsHalt;
					Process[m->pCfg->HeadCfg.TVL.PROC_Indx].xCMD = prcsHalt;
					Process[m->pCfg->HeadCfg.HW.PROC_Indx].xCMD = prcsHalt;
					Process[m->pCfg->HeadCfg.GAS.PROC_Indx].xCMD = prcsHalt;

				}

			}

		}
		ret = 2;

	TimerExecute(&CalibrTMR);

	if (m->CalibType == CALIB_NONE)
		ret = 0;

	return ret;
}

void IncrParam(CurCfg_typ * curCfg, UINT param, DINT segm, float gain)
{
int i;

	if (curCfg->Param[param].segmYes)
	{
		i = segm;

		if (i > SEGM_NUM_MAX)
			i = SEGM_NUM_MAX;
	}
	else
		i = 0;

	curCfg->Param[param].val[i] += curCfg->Param[param].incr * gain;

	if (curCfg->Param[param].val[i] > curCfg->Param[param].max)
		curCfg->Param[param].val[i] = curCfg->Param[param].max;

	return;

}

void DecrParam(CurCfg_typ * curCfg, UINT param, DINT segm, float gain)
{
	int i;

	if (curCfg->Param[param].segmYes)
	{
		i = segm;

		if (i > SEGM_NUM_MAX)
			i = SEGM_NUM_MAX;
	}
	else
		i = 0;

	curCfg->Param[param].val[i] -= curCfg->Param[param].incr * gain;

	if (curCfg->Param[param].val[i] < curCfg->Param[param].min)
		curCfg->Param[param].val[i] = curCfg->Param[param].min;

	return;
}

void Check_parOSC_Amplit(CurCfg_typ * curCfg, HMI_typ * hmi, UINT seg)
{
float x;
UINT _seg;

	if(curCfg->Param[parOSC_FinalAmplit].segmYes)
		_seg = seg;
	else
		_seg = 0;

	if(curCfg->Param[parOSC_Amplit].val[seg] < curCfg->Param[parOSC_FinalAmplit].val[_seg] ){

		curCfg->Param[parOSC_Amplit].val[seg] = curCfg->Param[parOSC_FinalAmplit].val[_seg];

		strcpy(hmi->pMessage[0], " OSC Primery	 ");
		strcpy(hmi->pMessage[1], " Amplitude ");
		strcpy(hmi->pMessage[2], " smaller then ");
		strcpy(hmi->pMessage[3], " Final Amplitude");
		TimerStart(&hmi->MsgTmr, 1.5);

	}

	if(curCfg->Param[parOSC_InitAmplit].segmYes)
		_seg = seg;
	else
		_seg = 0;

	if(curCfg->Param[parOSC_Amplit].val[seg] < curCfg->Param[parOSC_InitAmplit].val[_seg] ){

		curCfg->Param[parOSC_Amplit].val[seg] = curCfg->Param[parOSC_InitAmplit].val[_seg];

		strcpy(hmi->pMessage[0], " OSC Primery	 ");
		strcpy(hmi->pMessage[1], " Amplitude ");
		strcpy(hmi->pMessage[2], " smaller then ");
		strcpy(hmi->pMessage[3], " Init Amplitude");
		TimerStart(&hmi->MsgTmr, 1.5);

	}

	if (curCfg->Param[parOSC_Excur].val[seg] > 0)
	{

		x = curCfg->Param[parOSC_Amplit].val[seg] / curCfg->Param[parOSC_Excur].val[seg];

		if (x > curCfg->Param[parOSC_MaxTvlVel].val[0])
		{
			curCfg->Param[parOSC_Amplit].val[seg] =
			curCfg->Param[parOSC_MaxTvlVel].val[0] *curCfg->Param[parOSC_Excur].val[seg];

			strcpy(hmi->pMessage[0], " OSC	 ");
			strcpy(hmi->pMessage[1], " Amplitude ");
			strcpy(hmi->pMessage[2], " was");
			strcpy(hmi->pMessage[3], " too high");
			TimerStart(&hmi->MsgTmr, 1.5);
		}

	}
}

void Check_parOSC_Excur(CurCfg_typ * curCfg, HMI_typ * hmi, UINT seg)
{
float x;

	if ((curCfg->Param[parOSC_Excur].val[seg] > 0) && (curCfg->Param[parOSC_MaxTvlVel].val[0] > 0))
	{
		x = curCfg->Param[parOSC_Amplit].val[seg] / curCfg->Param[parOSC_Excur].val[seg];

		if (x > curCfg->Param[parOSC_MaxTvlVel].val[0])
		{
			curCfg->Param[parOSC_Excur].val[seg] =
			curCfg->Param[parOSC_Amplit].val[seg] / curCfg->Param[parOSC_MaxTvlVel].val[0];

			strcpy(hmi->pMessage[0], " OSC	 ");
			strcpy(hmi->pMessage[1], " Excurtion ");
			strcpy(hmi->pMessage[2], " was");
			strcpy(hmi->pMessage[3], " too small");
			TimerStart(&hmi->MsgTmr, 1.5);
		}

	}
	return;
}

void Fill_Segments(CurCfg_typ * curCfg, UINT par, UINT seg, UINT Mode, UINT Step)
{
float x;
int i;

	if (!curCfg->Param[par].segmYes)
		return;

	switch (Mode)
	{
		case 1:

			for (i = seg; i < SEGM_NUM_MAX; i++)
				curCfg->Param[par].val[i] = curCfg->Param[par].val[seg];

		break;

		case 2:

			if (Step == 51)
			{ // RUN
				for (i = seg; i < SEGM_NUM_MAX; i++)
					curCfg->Param[par].val[i] = curCfg->Param[par].val[seg];
			}

		break;

		default:
			// OFF
		break;
	}

	return;
}

void SetBannerTxt(MASTER_typ * m, HMI_typ * hmi, HMI_INTRF_typ * intrf)
{

	if (!m || !hmi || !intrf)
	return;

	if (!hmi->pBanner)
	return;

	if(m->sm.Step == 251){ // Head was changed

		strcpy(hmi->pBanner ,"Head Setup Changed - Must Restart!!!");

		return;

	}

	if(TVL_MAP_Step > 0)
		strcpy(hmi->pBanner ,"REC. ");
	else {

		if((curCalib->GenSetup[SETUP_EXTRAS]&0x1) != 0)
			strcpy(hmi->pBanner ,"Sup.//");
		else
			strcpy(hmi->pBanner ," ");

	}

	if((curCalib->GenSetup[SETUP_EXTRAS]&0x1) != 0){

		if(Weld_Report_Status == 2)
			strcat(hmi->pBanner , "W:Report !!!  ");

	}

	//strcpy(hmi->pBanner, "");

#ifdef UNIV_SYSTEM
	if (!Hardware[1].CouplerOK[0])
	{

#ifndef TEST_ONLY_PLC_ANDROID
		strcat(hmi->pBanner, "Ext. Suitcase Err ");
		return;

#endif

	}
	else
#endif

	if(m->sm.Step == 999){
		xsprintf(hmi->pBanner + strlen(hmi->pBanner)," TML Ref. Setup Finished - Restart Power ");
		return;
	}

	else if(m->sm.Step == 1000){
		xsprintf(hmi->pBanner + strlen(hmi->pBanner),"TML Setup Fin. Restart or Start New One ");
		return;
	}
	else if(m->sm.Step == 1001){
		xsprintf(hmi->pBanner + strlen(hmi->pBanner),"New Head Selected Restart Power ");
		return;
	}
	else if ((m->sm.Step >= 230) && (m->sm.Step <= 236)){

		switch (m->sm.Step)
		{

			case 230:

				xsprintf(hmi->pBanner + strlen(hmi->pBanner), "Clear ESTOP to Refresh TML Setup ");

			break;

			case 231:

				xsprintf(hmi->pBanner + strlen(hmi->pBanner), "Press START for TML Check ");

			break;

			case 232:

				xsprintf(hmi->pBanner + strlen(hmi->pBanner), "Wait!! Checking TML  %3.1f",  ((float) (m->sm.Tmr1.PT - m->sm.Tmr1.ET)) / 1000.0);

			break;

			case 233:

				xsprintf(hmi->pBanner + strlen(hmi->pBanner), "Press START Btn for %s  Setup Download " , TML_MTR_INST[curTML_indx].Name);

			break;

			case 234:
			case 235:
			case 236:

				xsprintf(hmi->pBanner + strlen(hmi->pBanner), "Wait!! TML Setup %s %d %3.1f", TML_MTR_INST[curTML_indx].Name, TML_MTR_INST[curTML_indx].xCMD, (float) m->sm.Tmr1.ET / 1000.0);

			break;

			default:

				xsprintf(hmi->pBanner + strlen(hmi->pBanner), "Wait!! Checking TML");

			break;
		}

		return;

	}
	else if ((VectorStateMach[VECT_TVL].FbkVect.Mode == vectSt_Mode_Vel) && VectorStateMach[VECT_TVL].FbkWarning)
	{
		if(VectorStateMach[VECT_TVL].FbkWarning == 2)
			strcat(hmi->pBanner, "Max Cmd TVL - slow down !!!");
		else
			strcat(hmi->pBanner, "TVL Limits are reached !!!");

		return;

	}
	else if ((ErrorMgr.Error != 0) && (!m->LOCKED))
	{

		switch (ErrorMgr.Error)
		{
			case ERROR_FATAL:
				strcat(hmi->pBanner, "FATAL ERR MUST RBT !!!");
			break;

			default:
				if((m->sm.Step == 191)
					||(m->sm.Step == 200)) // waiting ESTOP recovery
					strcat(hmi->pBanner, "Do NOT Hold BUTTON when clear error !!!");
				else
					strcat(hmi->pBanner, "	ERROR  !!!");
			break;
		}

		return;
	}
	else if (m->ESTOP)
	{

		if(m->pESTOP_Out){

			if(*m->pESTOP_Out)
				strcat(hmi->pBanner, " ESTOP !!! ");
			else
				strcat(hmi->pBanner, " ESTOP *** ");

		}
		else
			strcat(hmi->pBanner, " ESTOP !!! ");

		return;

	}
	else if (intrf->GlblBtnCmd[0])
	{

		strcat(hmi->pBanner, hmi->ActiveBanner);

		return;

	}

	switch (m->sm.Step)
	{

		case 1:

			xsprintf(hmi->pBanner , "Check TML Ax: %d  ", (DINT)TML_Restart_Indx);

		break;

		case 49:

			strcat(hmi->pBanner, "Wait for ArcLink");

		break;

		case 50:

			if ((Process[m->pCfg->HeadCfg.OSC.PROC_Indx].Status == prcsSTATUS_Stopped) ||
			(Process[m->pCfg->HeadCfg.OSC.PROC_Indx].Status == prcsSTATUS_DirectCntrl))
			{
				strcat(hmi->pBanner, "  STOP ");

				if(curCalib->GenSetup[SETUP_CONTIN_WELD] == 2)
					strcat(hmi->pBanner, "Cont.");
				else if(curCalib->GenSetup[SETUP_CONTIN_WELD] == 1)
					strcat(hmi->pBanner, "Cont. One Way");

			}
			else if (Process[m->pCfg->HeadCfg.OSC.PROC_Indx].Status == prcsSTATUS_Run)
				strcat(hmi->pBanner, " OSC Test ");

		break;

		case 51:

			switch (m->SeqStep)
				{
				case 1:

					xsprintf(hmi->pBanner + strlen(hmi->pBanner), "START !!! %3.1f ",((float) (m->sm.Tmr1.PT - m->sm.Tmr1.ET)) / 1000.0);

				break;

				case 2:

					strcat(hmi->pBanner, " Wait ARC ");

				break;

				case 3:

					strcat(hmi->pBanner, " RUN ");

					if(curCalib->GenSetup[SETUP_CONTIN_WELD]> 0){

						if(Cont_Stop_By_End)
							strcat(hmi->pBanner, "To STOP !!");
						else {

							if(curCalib->GenSetup[SETUP_CONTIN_WELD] == 2)
								strcat(hmi->pBanner, "Cont.");
							else
								strcat(hmi->pBanner, "Cont. One Way");

						}

					}

				break;

				case 150:

					xsprintf(hmi->pBanner + strlen(hmi->pBanner), "REWRAP !!! %3.1f ",	((float) (m->sm.Tmr1.PT - m->sm.Tmr1.ET)) / 1000.0);

				break;

				case 201:

					switch (Process[m->pCfg->HeadCfg.TVL.PROC_Indx].Status)
					{
						case prcsSTATUS_StopDly:
							strcat(hmi->pBanner, "TVL Stop Dly");
						break;

						case prcsSTATUS_RampDwn:
							strcat(hmi->pBanner, "TVL Ramp Dwn");
						break;

						case prcsSTATUS_ReturnDly:
							strcat(hmi->pBanner, "TVL Ret Dly");
						break;

						case prcsSTATUS_Return:
							strcat(hmi->pBanner, "TVL Return");
						break;

						default:
							strcat(hmi->pBanner, "Ramp Down");
						break;
					}

				break;

				case 202:

					strcat(hmi->pBanner, "Wait Index");

				break;

				case 203:

					strcat(hmi->pBanner, "Wait Head Return");

				break;

				case 205:

					strcat(hmi->pBanner, "Wait New File Load");

				break;

				case 210:

					strcat(hmi->pBanner, "Going to Start Pos.");

				break;

				case 220:

					xsprintf(hmi->pBanner + strlen(hmi->pBanner), "AUTO START !!! %3.1f ",	((float) (m->sm.Tmr1.PT - m->sm.Tmr1.ET)) / 1000.0);

				break;

				case 255:

					strcat(hmi->pBanner, "Wait OSC Stop");

				break;

				default:

					strcat(hmi->pBanner, " Stopping ");
					if(curCalib->GenSetup[SETUP_CONTIN_WELD]> 0){

						if(curCalib->GenSetup[SETUP_CONTIN_WELD] == 2)
							strcat(hmi->pBanner, "Cont.");
						else
							strcat(hmi->pBanner, "Cont. One Way");

						//strcat(hmi->pBanner, "Cont.");

					}

				break;
			}

		break;

		case 100:
			/*
			if(hmi->curHeadID < 0xFFFE)
				strcat (hmi->pBanner , hmi->ActiveBanner);
			else */
			strcat(hmi->pBanner, " Calib.STOP ");

		break;

		case 101:
			/*if(hmi->curHeadID < 0xFFFE)
				strcat (hmi->pBanner , hmi->ActiveBanner);
			else */
			strcat(hmi->pBanner, " Calib.RUN ");

		break;

		case 220:

			strcat(hmi->pBanner, " TML Firm. ");

		break;

		case 230:

			strcpy(hmi->pBanner, " NEW HEAD CONFIGURATION was Selected");

		break;

		default:

			//strcat(hmi->pBanner, " INIT ");
			strcat(hmi->pBanner, m->sm.Text);

		break;
	}

	switch (m->SubSeqStep)
	{
		default:
		break;

		case 1:
			strcat(hmi->pBanner, " >>T");
		break;

		case 2:
			strcat(hmi->pBanner, " >>R");
		break;
	}

	/*
	if(intrf->TestMode)
	strcat(hmi->pBanner , " TEST");

	if(m->WireDisabled)
	strcat(hmi->pBanner , "/WIRE OFF");

	if(Process[m->pCfg->HeadCfg.AVC.PROC_Indx].Param[0])
	strcat(hmi->pBanner , "/LOCKED");
	*/

	return;

}

float getBtnProgress()
{

	return (float) (btnProgress + btnProgressBias) / (float) (btnProgressMax + btnProgressBias);

}

void SetZeroPosition(MASTER_typ * m)
{
	curCalib->GenSetup[SETUP_ZIG_ZAG] = 0;

	if (TVL_ROT_Param_Set[0].pEncoder){
		OLD_MTR_POS[TVL_ZONE_HOME] = *TVL_ROT_Param_Set[0].pEncoder;

		Process[PROC_WRST].xCMD = prcsRetract;

	}

return;

}

void CreateParamList()
{
UINT i;

	i = 0;
	ParamList.Index[i++] = parGEN_WeldProgramRepeat;

	// All parameters from segment editor
	ParamList.Index[i++] = parTIG_AmpSP;
	ParamList.Index[i++] = parTIG_AmpInSP;
	ParamList.Index[i++] = parTIG_AmpOutSP;
	ParamList.Index[i++] = parTIG_BackAmp;
	ParamList.Index[i++] = parTIG_PulseFreq;
	ParamList.Index[i++] = parTIG_PulseWidth;

	ParamList.Index[i++] = parAVC_VoltSP;
	ParamList.Index[i++] = parAVC_VoltInSP;
	ParamList.Index[i++] = parAVC_VoltOutSP;
	ParamList.Index[i++] = parAVC_VoltBackSP;

	ParamList.Index[i++] = parTVL_VelSP;
	ParamList.Index[i++] = parTVL_VelInSP;
	ParamList.Index[i++] = parTVL_VelOutSP;
	ParamList.Index[i++] = parTVL_VelBackSP;

	ParamList.Index[i++] = parWF_SpeedSP;
	ParamList.Index[i++] = parWF_SpeedInSP;
	ParamList.Index[i++] = parWF_SpeedOutSP;
	ParamList.Index[i++] = parWF_BkgSpeedSP;

	ParamList.Index[i++] = parWP_SpeedSP;
	ParamList.Index[i++] = parWP_SpeedInSP;
	ParamList.Index[i++] = parWP_SpeedOutSP;
	ParamList.Index[i++] = parWP_BkgSpeedSP;

	ParamList.Index[i++] = parHW_AmpSP;
	ParamList.Index[i++] = parOSC_Amplit;
	ParamList.Index[i++] = parOSC_Excur;
	ParamList.Index[i++] = parOSC_Dwell_In;
	ParamList.Index[i++] = parOSC_Dwell_Out;

	// All parameters  from Timing Calculation
	ParamList.Index[i++] = parAVC_Upslope;
	ParamList.Index[i++] = parAVC_StopDly;
	ParamList.Index[i++] = parAVC_DownSlope;

	ParamList.Index[i++] = parTVL_StartDly;
	ParamList.Index[i++] = parTVL_RampUp;
	ParamList.Index[i++] = parTVL_StopDly;
	ParamList.Index[i++] = parTVL_RampDwn;
	ParamList.Index[i++] = parTVL_RewrapDly;
	ParamList.Index[i++] = parTVL_RunDist;
	ParamList.Index[i++] = parTVL_OverlapDist;

	ParamList.Index[i++] = parWF_StartDly;
	ParamList.Index[i++] = parWF_RampUp;
	ParamList.Index[i++] = parWF_StopDly;
	ParamList.Index[i++] = parWF_RampDwn;
	ParamList.Index[i++] = parWF_RetractDly;

	ParamList.Index[i++] = parTIG_StartDly;
	ParamList.Index[i++] = parTIG_RampUp;
	ParamList.Index[i++] = parTIG_StopDly;
	ParamList.Index[i++] = parTIG_RampDwn;

	ParamList.Index[i++] = parOSC_StartDly;
	ParamList.Index[i++] = parOSC_RampUp;
	ParamList.Index[i++] = parOSC_StopDly;
	ParamList.Index[i++] = parOSC_RampDwn;

	ParamList.Index[i++] = parWP_StartDly;
	ParamList.Index[i++] = parWP_RampUp;
	ParamList.Index[i++] = parWP_StopDly;
	ParamList.Index[i++] = parWP_RampDwn;

	ParamList.Index[i++] = parHW_RampUpDly;
	ParamList.Index[i++] = parHW_RampUp;
	ParamList.Index[i++] = parHW_RampDwnDly;
	ParamList.Index[i++] = parHW_RampDwn;
	ParamList.Index[i++] = parGAS_PostPurgeTm;

	ParamList.IndexNum	= i;

	i = 0;
	ParamList.Index_Enum[i++] = parENUM_WeldProgramLinkMode;
	ParamList.Index_Enum[i++] = parENUM_PathMode;
	//ParamList.Index_Enum[i++] = parENUM_WeldProgramCase;

	ParamList.IndexNum_Enum = i;

	i = 0;
	ParamList.Index_Int[i++] = parINT_NumZone;

	ParamList.IndexNum_Int = i;

}

void DeleteExtension(char * p)
{
UINT len, i;

	len = strlen(p);

	for (i = 0; i < len; i++)
	{
		if (p[i] == '.')
		{
			p[i]= 0;
			break;
		}
	}

	return;

}

void WireDisableInable(plcbit Tmr_Q)
{
	if (!m->WireDisabled)
	{

		if (Tmr_Q)
		{
			if ((Process[m->pCfg->HeadCfg.WP.PROC_Indx].Status == prcsSTATUS_Stopped)
				|| (Process[m->pCfg->HeadCfg.WP.PROC_Indx].Status == prcsSTATUS_Retract)
				|| (Process[m->pCfg->HeadCfg.WP.PROC_Indx].Status == prcsSTATUS_RampDwn)
				|| (Process[m->pCfg->HeadCfg.WP.PROC_Indx].Status == prcsSTATUS_StopDly)){

					switch(curCalib->GenSetup[SETUP_WF_RAMP] & 0x4){

						case 0:  // No Ramps

							Process[m->pCfg->HeadCfg.WP.PROC_Indx].xCMD = prcsJump2Run;

						break;

						default:

							Process[m->pCfg->HeadCfg.WP.PROC_Indx].Param[0] = 1; // Skip all delays - regular ramps
							Process[m->pCfg->HeadCfg.WP.PROC_Indx].xCMD = prcsQuickStart;

						break;
					}

			}

			if ((Process[m->pCfg->HeadCfg.WF.PROC_Indx].Status == prcsSTATUS_Stopped)
				|| (Process[m->pCfg->HeadCfg.WF.PROC_Indx].Status == prcsSTATUS_Retract)
				|| (Process[m->pCfg->HeadCfg.WF.PROC_Indx].Status == prcsSTATUS_RampDwn)
				|| (Process[m->pCfg->HeadCfg.WF.PROC_Indx].Status == prcsSTATUS_StopDly)){

					switch(curCalib->GenSetup[SETUP_WF_RAMP] & 0x4){

						case 0:  // No Ramps

							Process[m->pCfg->HeadCfg.WF.PROC_Indx].xCMD = prcsJump2Run;

						break;

						default:

							Process[m->pCfg->HeadCfg.WF.PROC_Indx].Param[0] = 1; // Skip all delays - regular ramps
							Process[m->pCfg->HeadCfg.WF.PROC_Indx].xCMD = prcsQuickStart;

						break;
					}

			}

			if (Process[m->pCfg->HeadCfg.HW.PROC_Indx].Status != prcsSTATUS_Run)
				Process[m->pCfg->HeadCfg.HW.PROC_Indx].xCMD = prcsJump2Run;

		}
		else
		{

			if(Process[m->pCfg->HeadCfg.WP.PROC_Indx].Status == prcsSTATUS_Stopped)
				Process[m->pCfg->HeadCfg.WP.PROC_Indx].xCMD = prcsSTART;

			if (Process[m->pCfg->HeadCfg.WF.PROC_Indx].Status == prcsSTATUS_Stopped)
				Process[m->pCfg->HeadCfg.WF.PROC_Indx].xCMD = prcsSTART;

			if (Process[m->pCfg->HeadCfg.HW.PROC_Indx].Status == prcsSTATUS_Stopped)
				Process[m->pCfg->HeadCfg.HW.PROC_Indx].xCMD = prcsSTART;

		}

	}
	else
	{

		if ((Process[m->pCfg->HeadCfg.WP.PROC_Indx].Status == prcsSTATUS_Run)
			|| (Process[m->pCfg->HeadCfg.WP.PROC_Indx].Status == prcsSTATUS_StartDly)
			|| (Process[m->pCfg->HeadCfg.WP.PROC_Indx].Status == prcsSTATUS_RampUp)){

			switch(curCalib->GenSetup[SETUP_WF_RAMP] & 0x3){

				case 0x0: // No ramp , no retract
				case 0x1: // No Ramp , Retract

					Process[m->pCfg->HeadCfg.WP.PROC_Indx].xCMD = prcsHalt;

				break;

				case 0x2: // Ramp , No Retract
				case 0x3: // Ramp , Retract

					Process[m->pCfg->HeadCfg.WP.PROC_Indx].Param[0] = 1; // Skip all delays , use ramp
					Process[m->pCfg->HeadCfg.WP.PROC_Indx].xCMD = prcsQuickSTOP;

				break;

			}
		}

		if ((Process[m->pCfg->HeadCfg.WF.PROC_Indx].Status == prcsSTATUS_Run)
			|| (Process[m->pCfg->HeadCfg.WF.PROC_Indx].Status == prcsSTATUS_StartDly)
			|| (Process[m->pCfg->HeadCfg.WF.PROC_Indx].Status == prcsSTATUS_RampUp)){

			switch(curCalib->GenSetup[SETUP_WF_RAMP] & 0x3){

				case 0x0: // No ramp , no retract

					Process[m->pCfg->HeadCfg.WF.PROC_Indx].xCMD = prcsHalt;

				break;

				case 0x1: // No Ramp , Retract

					Process[m->pCfg->HeadCfg.WF.PROC_Indx].Param[0] = 3; // Skip all delays , ramps , only retract
					Process[m->pCfg->HeadCfg.WF.PROC_Indx].xCMD = prcsQuickSTOP;

				break;

				case 0x2: // Ramp , No Retract

					Process[m->pCfg->HeadCfg.WF.PROC_Indx].Param[0] = 4; // Skip all delays , ramps , only retract
					Process[m->pCfg->HeadCfg.WF.PROC_Indx].xCMD = prcsQuickSTOP;

				break;

				case 0x3: // Ramp , Retract

					Process[m->pCfg->HeadCfg.WF.PROC_Indx].Param[0] = 1; // Skip all delays , use ramp
					Process[m->pCfg->HeadCfg.WF.PROC_Indx].xCMD = prcsQuickSTOP;

				break;

			}

		}

		if (Process[m->pCfg->HeadCfg.HW.PROC_Indx].Status != prcsSTATUS_Stopped)
			Process[m->pCfg->HeadCfg.HW.PROC_Indx].xCMD = prcsQuickSTOP;

	}

	return;
}

/*
prcsSTATUS_Retract
prcsSTATUS_RampDwn
prcsSTATUS_ReturnDly
prcsSTATUS_StopDly
*/

/* old one replaced 01 Apr2020
void WireDisableInable(plcbit Tmr_Q)
{
	if (!m->WireDisabled)
	{

		if (Tmr_Q)
		{
			if (Process[m->pCfg->HeadCfg.WP.PROC_Indx].Status == prcsSTATUS_Stopped)
				Process[m->pCfg->HeadCfg.WP.PROC_Indx].xCMD = prcsJump2Run;

			if (Process[m->pCfg->HeadCfg.WF.PROC_Indx].Status == prcsSTATUS_Stopped)
				Process[m->pCfg->HeadCfg.WF.PROC_Indx].xCMD = prcsJump2Run;

			if (Process[m->pCfg->HeadCfg.HW.PROC_Indx].Status == prcsSTATUS_Stopped)
				Process[m->pCfg->HeadCfg.HW.PROC_Indx].xCMD = prcsJump2Run;

		}
		else
		{

			if (Process[m->pCfg->HeadCfg.WP.PROC_Indx].Status == prcsSTATUS_Stopped)
				Process[m->pCfg->HeadCfg.WP.PROC_Indx].xCMD = prcsSTART;

			if (Process[m->pCfg->HeadCfg.WF.PROC_Indx].Status == prcsSTATUS_Stopped)
				Process[m->pCfg->HeadCfg.WF.PROC_Indx].xCMD = prcsSTART;

			if (Process[m->pCfg->HeadCfg.HW.PROC_Indx].Status == prcsSTATUS_Stopped)
				Process[m->pCfg->HeadCfg.HW.PROC_Indx].xCMD = prcsSTART;

		}

	}
	else
	{
		// Nowe
		if (Process[m->pCfg->HeadCfg.WP.PROC_Indx].Status == prcsSTATUS_Run)
			Process[m->pCfg->HeadCfg.WP.PROC_Indx].xCMD = prcsQuickSTOP;

		//Process[m->pCfg->HeadCfg.WP.PROC_Indx].xCMD = prcsHalt;
		if (Process[m->pCfg->HeadCfg.WF.PROC_Indx].Status != prcsSTATUS_Stopped) //Process[m->pCfg->HeadCfg.WF.PROC_Indx].xCMD = prcsHalt;
			Process[m->pCfg->HeadCfg.WF.PROC_Indx].xCMD = prcsQuickSTOP;

		if (Process[m->pCfg->HeadCfg.HW.PROC_Indx].Status != prcsSTATUS_Stopped)
			Process[m->pCfg->HeadCfg.HW.PROC_Indx].xCMD = prcsSTOP;

	}

	return;
}

*/

void DumpParamToFile()
{

char tmpTxt[32];
int len;

	switch (parametersDump_Step)
	{
		case 0:

		break;

		case 1:

			if (File_RW.CMD == 0)
			{

				strcpy(File_RW.deviceName, "WeldPrograms");
				File_RW._int.wStatus = 0;

				DTGetTime_1.enable	= 1;
				DTGetTime(&DTGetTime_1);
				DT_TO_DTStructure(DTGetTime_1.DT1, (UDINT) (&DTStruct));

				xsprintf(File_RW.fileNewName, "%s_%d_%d_%d.csv", curCfg->CurProgramName,
				DTStruct.hour, DTStruct.minute, DTStruct.second);

				File_RW._int.wStatus = 0;
				File_RW.CMD 		= F_OPEN_ONLY;
				parametersDump_Step++;

			}

		break;

		case 2:

			if (File_RW.CMD == 0)
			{

				File_RW.pMem		= (UDINT)
				LineTxt;
				File_RW.Offset		= 0;
				File_RW.Len 		= 0;

				//paramIndx			= parOSC_StartDly;
				paramIndx			= parLCD_BtnMode;

				/* status (20708 -> File doesn't exist) */
				if (File_RW._int.wStatus == 20708)
				{
					File_RW.CMD 		= F_CREATE_ONLY;
					parametersDump_Step++;
				}
				else if (!File_RW.Error)
				{
					File_RW.CMD 		= F_DELETE;
				}
				else
					parametersDump_Step = 0;

			}

		break;

		case 3:

			if (File_RW.CMD == 0)
			{
				ascDTStructure((UDINT) &DTStruct, tmpTxt, 25);

				xsprintf(LineTxt, " Program: %s -  Stored at: %s \n\n\r////// Parameters ///// \n\r  ",	curCfg->CurProgramName, tmpTxt);

				//ascDTStructure((UDINT) &DTStruct, LineTxt + strlen(LineTxt), 25);
				len = strlen(LineTxt);

				//LineTxt[len++]= 0x0D; //CR
				//LineTxt[len++]= 0x0D; // CR
				File_RW.Len 		= strlen(LineTxt);
				File_RW.CMD 		= F_WRITE_ONLY;
				parametersDump_Step++;

			}

		break;

		case 4:

			if (File_RW.CMD == 0)
			{

				if (paramIndx < parLAST_PARAM)
				{

					File_RW.Offset		+= File_RW.Len;

					if (strlen(cfg->ScaledVar[paramIndx].name) > 0)
					{
						xsprintf(LineTxt, "Par. %d ,   (%s) , [ %s ] = %s \n\r ", paramIndx, cfg->ScaledVar[paramIndx].enumTXT, cfg->ScaledVar[paramIndx].name, GetScaledVal(lcd, &cfg->ScaledVar[paramIndx], 0));
					}
					else
						xsprintf(LineTxt, "Par. %d:///	available\n\r ", paramIndx);

					File_RW.Len 		= strlen(LineTxt);
					File_RW.CMD 		= F_WRITE_ONLY;
					paramIndx++;

				}
				else
				{
					File_RW.Offset		+= File_RW.Len;

					xsprintf(LineTxt, "//////  Text Resources	///////// \n\r");
					File_RW.Len 		= strlen(LineTxt);
					File_RW.CMD 		= F_WRITE_ONLY;

					paramIndx			= 0;
					parametersDump_Step++;
				}

			}

		break;

		case 5:

			if (File_RW.CMD == 0)
			{

				if (paramIndx < TXT_RESOURCES_MAX)
				{
					if (strlen(cfg->TXT_Resources[paramIndx]) > 0)
					{

						File_RW.Offset		+= File_RW.Len;
						xsprintf(LineTxt, "Txt Res. %d , [ %s ] \n\r", paramIndx, cfg->TXT_Resources[paramIndx]);

						File_RW.Len 		= strlen(LineTxt);
						File_RW.CMD 		= F_WRITE_ONLY;

					}

					paramIndx++;
				}
				else
				{
					File_RW.Offset		+= File_RW.Len;

					xsprintf(LineTxt, "//////	Error Text	 ///////// \n\r");
					File_RW.Len 		= strlen(LineTxt);
					File_RW.CMD 		= F_WRITE_ONLY;

					paramIndx			= 0;
					parametersDump_Step++;

				}

			}

		break;

		case 6:

			if (File_RW.CMD == 0)
			{
				if (paramIndx < 128)
				{
					if (strlen(ErrorMgr.logs[paramIndx].txt) > 0)
					{
						File_RW.Offset		+= File_RW.Len;
						xsprintf(LineTxt, "Err %d , [ %s ] \n\r", paramIndx, ErrorMgr.logs[paramIndx].txt);

						File_RW.Len 		= strlen(LineTxt);
						File_RW.CMD 		= F_WRITE_ONLY;
					}

						paramIndx++;
					}
				else
				{

					paramIndx			= 0;
					parametersDump_Step = 10;

				}

			}

		break;

		case 10:

			File_RW.CMD = F_CLOSE_ONLY;
			parametersDump_Step = 0;

		break;

	}

}

void TVL_Map_ToFile()
{

char tmpTxt[32];
int len;

	switch (TVL_MAP_Step)
	{
		case 0:

			if(KK_HomeBtn)
				TVL_MAP_Step++;

		break;

		case 1:

			if (File_RW.CMD == 0)
			{

				strcpy(File_RW.deviceName, "TEMP");
				File_RW._int.wStatus = 0;

				DTGetTime_1.enable	= 1;
				DTGetTime(&DTGetTime_1);
				DT_TO_DTStructure(DTGetTime_1.DT1, (UDINT) (&DTStruct));

				xsprintf(File_RW.fileNewName, "TVL_MAP_%d_%d_%d.csv", DTStruct.hour, DTStruct.minute, DTStruct.second);

				File_RW._int.wStatus = 0;
				//File_RW.CMD 		= F_OPEN_ONLY;
				File_RW.CMD 		= F_CREATE_ONLY;
				//TVL_MAP_Step++;
				TVL_MAP_Step = 3;

			}

		break;

		case 2:

			if (File_RW.CMD == 0)
			{

				File_RW.pMem		= (UDINT)LineTxt;
				File_RW.Offset		= 0;
				File_RW.Len 		= 0;

				/* status (20708 -> File doesn't exist) */
				if (File_RW._int.wStatus == 20708)
				{
					File_RW.CMD 		= F_CREATE_ONLY;
					TVL_MAP_Step++;
				}
				else if (!File_RW.Error)
				{
					File_RW.CMD 		= F_DELETE;
				}
				else
					TVL_MAP_Step = 0;

			}

		break;

		case 3:

			if (File_RW.CMD == 0)
			{

				File_RW.pMem		= (UDINT)LineTxt;
				File_RW.Offset		= 0;
				File_RW.Len 		= 0;

				ascDTStructure((UDINT) &DTStruct, tmpTxt, 25);

				xsprintf(LineTxt, " TVL Mapping : Stored at: %s \n\n\r Id , Tick , TVL Set Speed , Mtr Delta , Encoder Delta  \n\r  ", tmpTxt);
				len = strlen(LineTxt);

				File_RW.Len 		= strlen(LineTxt);
				File_RW.CMD 		= F_WRITE_ONLY;

				TVL_MAP_Indx[0]		= 0;
				TVL_MAP_Indx_New[0] = 0;
				TVL_MAP_Step++;

			}

		break;

		case 4:

			if(KK_StopBtn)
				TVL_MAP_Step = 10;

			else if (File_RW.CMD == 0)
			{

				if (TVL_MAP_Indx_New[0])
				{

					TVL_MAP_Indx_New[0] = 0;

					File_RW.Offset		+= File_RW.Len;		//TVL_MAP_Indx[0], m->curSegm[ZONE]

					//xsprintf(LineTxt, " %d,%d, %4.2f ,%d,%d,%d\n ", TVL_MAP_Indx[0] ,actTicks , VectorStateMach[VECT_TVL].InVal ,  AxisCh[TML_AX_TVL].curPos , _deltaAPOS[0] , _deltaAPOS2[0]  );
					xsprintf(LineTxt, " %d,%d, %4.2f ,%d,%d\n ", TVL_MAP_Indx[0] ,actTicks , VectorStateMach[VECT_TVL].InVal  , _deltaAPOS[0] , _deltaAPOS2[0]  );
					//xsprintf(LineTxt, " %d,%d,%d,%d,%d\n\r ", TVL_MAP_Indx[0], m->curSegm[ZONE]  ,  AxisCh[TML_AX_TVL].curPos , _deltaAPOS[0] , _deltaAPOS2[0]  );
					File_RW.Len 		= strlen(LineTxt);
					File_RW.CMD 		= F_WRITE_ONLY;

				}
			}

		break;

		case 10:

			File_RW.CMD = F_CLOSE_ONLY;
			TVL_MAP_Step = 0;

		break;

	}

}

void EvaluatePosition()
{int type;

	 //VERSION with encoder

	//tickEncoder = (AxisCh[m->pCfg->HeadCfg.TVL.TML_Indx].curPos  - encHome);
	tickEncoder = (VectorStateMach[m->pCfg->HeadCfg.TVL.VECT_Indx].actPosDINT - OLD_MTR_POS[TVL_ZONE_HOME]);

	if(m->pCfg->HeadCfg.TVL.EncScale != 0.0){

		//ABS_TVL_Pos = (float)(tickEncoder * m->pCfg->HeadCfg.TVL.EncDenominator) / m->pCfg->HeadCfg.TVL.EncNominator;

		ABS_TVL_Pos = (float)((double)tickEncoder * m->pCfg->HeadCfg.TVL.EncScale);

		// Tak bylo przed 4 June 2021
		//actTicks = (DINT)ABS_TVL_Pos;

		if(TVL_ROT_Param_Set[0].EncPerTick > 0)
			actTicks = (DINT)((tickEncoder / TVL_ROT_Param_Set[0].EncPerTick)+0.5);
		else
			actTicks = (DINT)(ABS_TVL_Pos +0.5);

		actTicks = actTicks * m->pCfg->HeadCfg.TVL.Enc_Dir;

	}
	else { //old code

		if(TVL_ROT_Param_Set[0].EncPerTick > 0)
			actTicks = (DINT)(tickEncoder / TVL_ROT_Param_Set[0].EncPerTick);

		actTicks = actTicks * m->pCfg->HeadCfg.TVL.Enc_Dir;

		ABS_TVL_Pos = (float)tickEncoder / TVL_ROT_Param_Set[0].EncPerTick;

	}

	if (m->ticksPerSegm < 1)
		m->ticksPerSegm = 1;

	if (m->ticksPerZone < 1)
		m->ticksPerZone = 1;

	if(m->pCfg->HeadCfg.TVL.PinsPerRot) // static configuration
		curCalib->GenSetup[SETUP_PIN_PER_ROT] = m->pCfg->HeadCfg.TVL.PinsPerRot;

	m->curSegm[ACT_TVL_DIST] = TVL_ROT_Param_Set[0].EncPos_FBK;

	if(curCalib->GenSetup[SETUP_PIN_PER_ROT] > 0)
		actRot = actTicks / curCalib->GenSetup[SETUP_PIN_PER_ROT];

	//m->curSegm[FR_SEGM] = (actTicks / m->ticksPerSegm);
	//m->curSegm[HEAD_SEGM] = m->curSegm[ACT_TVL_DIST] / m->ticksPerSegm;

	actTicksForZone = actTicks;
	//actTicksForZone = KK_ActEnc;

	// Zone Position depends on head direction
	if (!m->ToolHeadID){

	}
	else
	{

		switch (curCalib->GenSetup[SETUP_TWO_TORCH])
		{
			default: // One Torch
				actTicksForZone = actTicksForZone *(-1);
			break;

			case 1: // Two Torches
				actTicksForZone = (curCalib->GenSetup[SETUP_PIN_PER_ROT] / 2) -actTicksForZone; // shift by 180 deg
			break;
		}

	}

	//////////////////////////////////////////////////

	switch(curCalib->GenSetup[SETUP_TWO_UP]){

		case 0: // One Up

			type = 0;

		break;

		case 1:

			if(curCalib->GenSetup[SETUP_ZONE_CENTR])
				type = 2; //  Gravity Centric
			else
				type = 1; // Start segm Centric

		break;

	}

	// KK - sprawdzic czy to cos pieprzy
	if(m->numZone <= 0)
		m->numZone = 1;

	if(curCalib->GenSetup[SETUP_PIN_PER_ROT] <= 0)
		curCalib->GenSetup[SETUP_PIN_PER_ROT] = 1;

	switch(type){

		case 0: // One Up

			m->ticksPerZone = (INT)(ceilf((float)curCalib->GenSetup[SETUP_PIN_PER_ROT]/(float)m->numZone));

			actTicksForZone = actTicksForZone%curCalib->GenSetup[SETUP_PIN_PER_ROT];
			if(actTicksForZone < 0)
				actTicksForZone += curCalib->GenSetup[SETUP_PIN_PER_ROT];

			m->curSegm[ZONE] = actTicksForZone / m->ticksPerZone;

		break;

		case 1: // Two up - Star Segment Centric

			m->ticksPerZone = (INT)(ceilf((float)curCalib->GenSetup[SETUP_PIN_PER_ROT]/((float)m->numZone * 2.0)));

				actTicksForZone = (actTicksForZone)%(curCalib->GenSetup[SETUP_PIN_PER_ROT]);
				if(actTicksForZone < 0)
					actTicksForZone += curCalib->GenSetup[SETUP_PIN_PER_ROT];

				m->curSegm[ZONE] = actTicksForZone / (m->ticksPerZone);

				m->curSegm[ZONE_RAW] = m->curSegm[ZONE] ;

				if(m->curSegm[ZONE] >= m->numZone )
					m->curSegm[ZONE] = (m->numZone * 2 -1) - m->curSegm[ZONE];

		break;

		case 2: // Two up - Gravity Centric

			if(m->numZone < 2.0)
				m->curSegm[ZONE] = 1;

			else {
				m->ticksPerZone = (INT)(ceilf((float)curCalib->GenSetup[SETUP_PIN_PER_ROT]/((float)m->numZone * 2.0 - 2.0)));

				actTicksForZone = (actTicksForZone + m->ticksPerZone/2)%(curCalib->GenSetup[SETUP_PIN_PER_ROT]);
				if(actTicksForZone < 0)
					actTicksForZone += curCalib->GenSetup[SETUP_PIN_PER_ROT];

				m->curSegm[ZONE] = actTicksForZone / (m->ticksPerZone);

				m->curSegm[ZONE_RAW] = m->curSegm[ZONE] ;

				if(m->curSegm[ZONE] >= m->numZone )
					m->curSegm[ZONE] = (m->numZone * 2 - 2) - m->curSegm[ZONE];

			}

		break;

	}

	if (m->curSegm[ZONE] < 0)
		m->curSegm[ZONE] = 0;;

	m->curSegm[ZONE] ++;

	////////////////////////
	if (m->curSegm[ZONE] > m->numZone)
		m->curSegm[ZONE] = m->numZone;

	//////////Zone calculating from Mapping /////////////
	//(curCalib->GenSetup[SETUP_MAPPING_ON] > 0)? 1:0;

	if(curCalib->GenSetup[SETUP_MAPPING_ON] != _MappingActive)
		PleaseUpdateHeadSetup(m);

	if((curCalib->GenSetup[SETUP_MAPPING_ON]&MAPPING_SEGM)){

		if(curCalib->GenSetup[SETUP_POLE_ELEMENTS] < 2)
			curCalib->GenSetup[SETUP_POLE_ELEMENTS] = 2;

		else if(curCalib->GenSetup[SETUP_POLE_ELEMENTS] > 32)
			curCalib->GenSetup[SETUP_POLE_ELEMENTS] = 32;

		m->numZone = curCalib->GenSetup[SETUP_POLE_ELEMENTS] * 2;
		m->curSegm[ZONE] = WRST_TML_Param_Set[0].actIndx +1;

	}

	_MappingActive = curCalib->GenSetup[SETUP_MAPPING_ON];

	//////////////////////////////////////////
	actTicksPerm = actTicks;

}

int WatchArcLinkError(MASTER_typ * m, Robot_typ * robot)
{
	int ret 			= 0;

	if(robot)
	{ // Arclink connection

		if(robot->Cntrl.Fbk.Error)
		{
			if(robot->Cntrl.Fbk.Error & ArcLink_Com_Failed){

				Errors(&ErrorMgr, ERROR_TIG_PROC, ERROR_ARCLINK_COM_LOST, (UDINT) robot->Cntrl.Fbk.Error);
				LogTxt(&LogMgr, "Arclink Com Err %d", (UDINT) robot->Cntrl.Fbk.Error);

			}else{

				Errors(&ErrorMgr, ERROR_TIG_PROC, ERROR_ARCLINK_PS_ERR, (UDINT) robot->Cntrl.Fbk.Error);
				LogTxt(&LogMgr, "Arclink Err %d", (UDINT) robot->Cntrl.Fbk.Error);

			}

			ret = 1;

		}

	}

	return ret;
}

void ChangeSegmentList(){
UINT _TVL_MODE , _WF_MODE , _WP_MODE;

	if(!curCfg)
		return;
	//////////////////////////////////////////

	if((curCfg->Param_ENUM[parENUM_TIG_Mode].val[0] != _TIG_Mode)
	|| (curCfg->Param_ENUM[parENUM_AVC_Mode].val[0] != _AVC_Mode)
	||(_TVL_SYN_MODE != curCfg->Param_ENUM[parENUM_TVL_SYN_MODE].val[0])
	||(_WF_SYN_MODE != curCfg->Param_ENUM[parENUM_WF_SYN_MODE].val[0])
	||(_WP_SYN_MODE != curCfg->Param_ENUM[parENUM_WP_SYN_MODE].val[0])
	){

		if(TVL_ROT_Param_Set[0].pSynchMode)
			_TVL_MODE = curCfg->Param_ENUM[parENUM_TVL_SYN_MODE].val[0];
		else
			_TVL_MODE = 0;

		if(WIRE_Param_Set[0].pSynchMode)
			_WF_MODE = curCfg->Param_ENUM[parENUM_WF_SYN_MODE].val[0];
		else
			_WF_MODE = 0;

		if(WIRE_Param_Set[1].pSynchMode)
			_WP_MODE = curCfg->Param_ENUM[parENUM_WP_SYN_MODE].val[0];
		else
			_WP_MODE = 0;

		switch(curCfg->Param_ENUM[parENUM_TIG_Mode].val[0]){

			default: // Straight

				curCfg->Param[parTIG_AmpSP].segmYes = 1;
				curCfg->Param[parTIG_AmpInSP].segmYes = 0;
				curCfg->Param[parTIG_AmpOutSP].segmYes = 0;
				curCfg->Param[parTIG_BackAmp].segmYes = 0;
				curCfg->Param[parTIG_PulseFreq].segmYes = 0;
				curCfg->Param[parTIG_PulseWidth].segmYes = 0;

				curCfg->Param[parAVC_VoltSP].segmYes = 1;
				curCfg->Param[parAVC_VoltInSP].segmYes = 0;
				curCfg->Param[parAVC_VoltOutSP].segmYes = 0;
				curCfg->Param[parAVC_VoltBackSP].segmYes = 0;

				/*
				curCfg->Param[parTVL_VelSP].segmYes = 1;
				curCfg->Param[parTVL_VelInSP].segmYes = 0;
				curCfg->Param[parTVL_VelOutSP].segmYes = 0;
				curCfg->Param[parTVL_VelBackSP].segmYes = 0;

				curCfg->Param[parWP_SpeedSP].segmYes = 1;
				curCfg->Param[parWP_SpeedInSP].segmYes = 0;
				curCfg->Param[parWP_SpeedOutSP].segmYes = 0;
				curCfg->Param[parWP_BkgSpeedSP].segmYes = 0;

				curCfg->Param[parWF_SpeedSP].segmYes = 1;
				curCfg->Param[parWF_SpeedInSP].segmYes = 0;
				curCfg->Param[parWF_SpeedOutSP].segmYes = 0;
				curCfg->Param[parWF_BkgSpeedSP].segmYes = 0;
				*/
```
